C03599=1044.445,262.335,-106.667,171.686,39.912,157.590
C03600=1044.439,262.088,-106.637,171.684,39.910,157.589
C03601=1044.432,261.839,-106.607,171.681,39.908,157.589
C03602=1044.425,261.591,-106.577,171.677,39.906,157.588
C03603=1044.419,261.343,-106.548,171.675,39.903,157.587
C03604=1044.411,261.094,-106.518,171.672,39.901,157.587
C03605=1044.405,260.847,-106.488,171.669,39.898,157.586
C03606=1044.398,260.598,-106.459,171.666,39.896,157.586
C03607=1044.391,260.351,-106.429,171.663,39.894,157.585
C03608=1044.385,260.102,-106.400,171.661,39.892,157.584
C03609=1044.378,259.854,-106.370,171.658,39.889,157.584
C03610=1044.371,259.605,-106.341,171.654,39.887,157.583
C03611=1044.365,259.358,-106.311,171.652,39.885,157.583
C03612=1044.358,259.109,-106.282,171.649,39.882,157.582
C03613=1044.351,258.862,-106.252,171.646,39.880,157.581
C03614=1044.344,258.613,-106.222,171.643,39.878,157.581
C03615=1044.337,258.365,-106.194,171.640,39.876,157.580
C03616=1044.330,258.117,-106.164,171.638,39.873,157.580
C03617=1044.324,257.869,-106.135,171.635,39.871,157.579
C03618=1044.317,257.620,-106.105,171.632,39.868,157.578
C03619=1044.311,257.372,-106.076,171.629,39.866,157.578
C03620=1044.304,257.124,-106.047,171.626,39.864,157.577
C03621=1044.297,256.876,-106.016,171.624,39.862,157.577
C03622=1044.291,256.628,-105.987,171.621,39.859,157.576
C03623=1044.284,256.379,-105.958,171.618,39.857,157.575
C03624=1044.277,256.131,-105.928,171.615,39.855,157.575
C03625=1044.271,255.883,-105.899,171.612,39.852,157.574
C03626=1044.264,255.634,-105.870,171.610,39.850,157.573
C03627=1044.258,255.387,-105.840,171.607,39.848,157.573
C03628=1044.251,255.138,-105.811,171.604,39.845,157.572
C03629=1044.245,254.890,-105.782,171.602,39.843,157.572
C03630=1044.238,254.642,-105.753,171.598,39.841,157.571
C03631=1044.231,254.394,-105.723,171.595,39.838,157.570
C03632=1044.224,254.146,-105.694,171.593,39.836,157.570
C03633=1044.218,253.898,-105.665,171.590,39.834,157.569
C03634=1044.211,253.649,-105.636,171.588,39.831,157.569
C03635=1044.205,253.401,-105.606,171.585,39.829,157.568
C03636=1044.198,253.153,-105.577,171.583,39.827,157.567
C03637=1044.192,252.904,-105.547,171.579,39.824,157.567
C03638=1044.185,252.656,-105.518,171.576,39.822,157.566
C03639=1044.179,252.408,-105.489,171.574,39.820,157.566
C03640=1044.171,252.160,-105.460,171.571,39.817,157.565
C03641=1044.165,251.912,-105.431,171.568,39.815,157.564
C03642=1044.159,251.664,-105.402,171.566,39.812,157.564
C03643=1044.152,251.416,-105.373,171.563,39.810,157.563
C03644=1044.146,251.167,-105.343,171.561,39.808,157.563
C03645=1044.139,250.919,-105.314,171.557,39.806,157.562
C03646=1044.133,250.671,-105.285,171.554,39.803,157.561
C03647=1044.126,250.422,-105.256,171.552,39.801,157.561
C03648=1044.120,250.174,-105.227,171.549,39.798,157.560
C03649=1044.113,249.926,-105.198,171.546,39.796,157.560
C03650=1044.107,249.678,-105.169,171.544,39.794,157.559
C03651=1044.100,249.430,-105.140,171.541,39.791,157.558
C03652=1044.093,249.147,-105.106,171.539,39.789,157.558
C03653=1044.085,248.864,-105.074,171.535,39.786,157.557
C03654=1044.078,248.581,-105.040,171.532,39.784,157.556
C03655=1044.071,248.298,-105.008,171.530,39.781,157.556
C03656=1044.064,248.050,-104.978,171.527,39.778,157.555
C03657=1044.058,247.802,-104.949,171.523,39.776,157.554
C03658=1044.052,247.554,-104.920,171.521,39.773,157.554
C03659=1044.046,247.305,-104.891,171.518,39.771,157.553
C03660=1044.039,247.057,-104.862,171.515,39.769,157.553
C03661=1044.032,246.809,-104.834,171.513,39.767,157.552
C03662=1044.025,246.561,-104.804,171.510,39.764,157.551
C03663=1044.019,246.313,-104.775,171.508,39.762,157.551
C03664=1044.013,246.064,-104.746,171.505,39.759,157.550
C03665=1044.007,245.816,-104.718,171.502,39.757,157.550
C03666=1044.001,245.568,-104.689,171.500,39.755,157.549
C03667=1043.994,245.320,-104.661,171.497,39.752,157.548
C03668=1043.987,245.071,-104.631,171.495,39.750,157.548
C03669=1043.981,244.823,-104.602,171.492,39.747,157.547
C03670=1043.974,244.574,-104.574,171.489,39.745,157.547
C03671=1043.968,244.326,-104.545,171.487,39.743,157.546
C03672=1043.961,244.078,-104.516,171.484,39.741,157.545
C03673=1043.955,243.830,-104.489,171.482,39.738,157.545
C03674=1043.949,243.581,-104.460,171.479,39.736,157.544
C03675=1043.941,243.333,-104.431,171.477,39.734,157.544
C03676=1043.935,243.085,-104.402,171.474,39.731,157.543
C03677=1043.929,242.836,-104.373,171.471,39.729,157.542
C03678=1043.922,242.588,-104.345,171.469,39.726,157.542
C03679=1043.916,242.340,-104.317,171.466,39.724,157.541
C03680=1043.909,242.092,-104.288,171.464,39.722,157.541
C03681=1043.903,241.844,-104.259,171.461,39.720,157.540
C03682=1043.896,241.595,-104.231,171.458,39.717,157.539
C03683=1043.890,241.347,-104.202,171.456,39.715,157.539
C03684=1043.883,241.099,-104.173,171.453,39.713,157.538
C03685=1043.876,240.850,-104.145,171.451,39.711,157.538
C03686=1043.869,240.602,-104.117,171.448,39.708,157.537
C03687=1043.863,240.353,-104.088,171.445,39.706,157.537
C03688=1043.856,240.105,-104.060,171.443,39.704,157.536
C03689=1043.850,239.857,-104.032,171.440,39.701,157.535
C03690=1043.844,239.608,-104.004,171.438,39.699,157.535
C03691=1043.837,239.360,-103.976,171.435,39.696,157.534
C03692=1043.830,239.112,-103.948,171.432,39.694,157.534
C03693=1043.824,238.864,-103.919,171.430,39.692,157.533
C03694=1043.817,238.615,-103.891,171.427,39.690,157.532
C03695=1043.810,238.367,-103.863,171.425,39.687,157.532
C03696=1043.804,238.119,-103.834,171.422,39.685,157.531
C03697=1043.797,237.870,-103.806,171.420,39.683,157.531
C03698=1043.790,237.622,-103.778,171.417,39.680,157.530
C03699=1043.784,237.373,-103.749,171.415,39.678,157.530
C03700=1043.777,237.125,-103.721,171.413,39.676,157.529
C03701=1043.770,236.877,-103.693,171.410,39.674,157.528
C03702=1043.764,236.628,-103.665,171.408,39.671,157.528
C03703=1043.757,236.380,-103.636,171.405,39.669,157.527
C03704=1043.751,236.132,-103.609,171.403,39.667,157.527
C03705=1043.744,235.883,-103.581,171.400,39.665,157.526
C03706=1043.738,235.635,-103.553,171.397,39.662,157.526
C03707=1043.731,235.387,-103.524,171.395,39.660,157.525
C03708=1043.724,235.098,-103.492,171.392,39.657,157.524
C03709=1043.716,234.809,-103.459,171.390,39.655,157.524
C03710=1043.708,234.520,-103.427,171.386,39.652,157.523
C03711=1043.701,234.232,-103.394,171.383,39.649,157.522
C03712=1043.695,233.984,-103.366,171.381,39.647,157.522
C03713=1043.688,233.736,-103.339,171.378,39.645,157.521
C03714=1043.681,233.488,-103.310,171.377,39.642,157.521
C03715=1043.675,233.239,-103.282,171.374,39.640,157.520
C03716=1043.668,232.991,-103.254,171.371,39.638,157.519
C03717=1043.662,232.742,-103.226,171.369,39.635,157.519
C03718=1043.655,232.494,-103.199,171.366,39.633,157.518
C03719=1043.649,232.245,-103.170,171.364,39.631,157.518
C03720=1043.642,231.997,-103.142,171.361,39.629,157.517
C03721=1043.635,231.749,-103.114,171.359,39.626,157.517
C03722=1043.629,231.500,-103.086,171.357,39.624,157.516
C03723=1043.622,231.252,-103.059,171.354,39.622,157.515
C03724=1043.615,231.003,-103.031,171.352,39.619,157.515
C03725=1043.609,230.756,-103.004,171.349,39.617,157.514
C03726=1043.603,230.507,-102.976,171.347,39.615,157.514
C03727=1043.597,230.258,-102.947,171.344,39.613,157.513
C03728=1043.590,230.010,-102.920,171.342,39.610,157.513
C03729=1043.583,229.762,-102.892,171.340,39.608,157.512
C03730=1043.577,229.513,-102.864,171.337,39.606,157.512
C03731=1043.570,229.265,-102.837,171.335,39.603,157.511
C03732=1043.563,229.016,-102.809,171.332,39.601,157.510
C03733=1043.557,228.768,-102.781,171.330,39.599,157.510
C03734=1043.550,228.520,-102.754,171.327,39.597,157.509
C03735=1043.544,228.272,-102.726,171.325,39.594,157.509
C03736=1043.537,228.023,-102.698,171.323,39.592,157.508
C03737=1043.530,227.775,-102.671,171.321,39.590,157.508
C03738=1043.524,227.526,-102.644,171.318,39.587,157.507
C03739=1043.517,227.277,-102.616,171.315,39.585,157.506
C03740=1043.511,227.029,-102.588,171.313,39.583,157.506
C03741=1043.503,226.781,-102.561,171.310,39.581,157.505
C03742=1043.497,226.533,-102.534,171.309,39.578,157.505
C03743=1043.491,226.284,-102.506,171.306,39.576,157.504
C03744=1043.484,226.035,-102.479,171.304,39.574,157.504
C03745=1043.477,225.787,-102.451,171.301,39.571,157.503
C03746=1043.471,225.539,-102.423,171.298,39.569,157.502
C03747=1043.464,225.290,-102.396,171.297,39.567,157.502
C03748=1043.457,225.042,-102.368,171.294,39.564,157.501
C03749=1043.451,224.794,-102.342,171.292,39.562,157.501
C03750=1043.444,224.545,-102.314,171.289,39.560,157.500
C03751=1043.438,224.297,-102.286,171.287,39.558,157.500
C03752=1043.431,224.048,-102.259,171.285,39.555,157.499
C03753=1043.424,223.799,-102.232,171.283,39.553,157.498
C03754=1043.418,223.551,-102.204,171.280,39.551,157.498
C03755=1043.412,223.303,-102.177,171.277,39.548,157.497
C03756=1043.405,223.054,-102.150,171.275,39.546,157.497
C03757=1043.398,222.806,-102.122,171.273,39.544,157.496
C03758=1043.392,222.558,-102.095,171.271,39.541,157.496
C03759=1043.385,222.309,-102.068,171.268,39.539,157.495
C03760=1043.379,222.061,-102.040,171.266,39.537,157.495
C03761=1043.372,221.812,-102.013,171.264,39.534,157.494
C03762=1043.366,221.564,-101.986,171.262,39.532,157.493
C03763=1043.360,221.315,-101.958,171.259,39.530,157.493
C03764=1043.352,221.020,-101.926,171.256,39.527,157.492
C03765=1043.344,220.723,-101.893,171.254,39.524,157.491
C03766=1043.336,220.427,-101.861,171.251,39.522,157.491
C03767=1043.329,220.131,-101.829,171.248,39.519,157.490
C03768=1043.321,219.883,-101.802,171.246,39.517,157.490
C03769=1043.315,219.634,-101.775,171.243,39.514,157.489
C03770=1043.308,219.386,-101.748,171.242,39.512,157.488
C03771=1043.302,219.137,-101.721,171.239,39.510,157.488
C03772=1043.295,218.889,-101.693,171.237,39.507,157.487
C03773=1043.288,218.640,-101.667,171.234,39.505,157.487
C03774=1043.282,218.392,-101.639,171.233,39.503,157.486
C03775=1043.275,218.144,-101.613,171.230,39.500,157.486
C03776=1043.268,217.895,-101.586,171.227,39.498,157.485
C03777=1043.262,217.646,-101.558,171.226,39.496,157.485
C03778=1043.255,217.398,-101.532,171.223,39.493,157.484
C03779=1043.248,217.150,-101.504,171.221,39.492,157.484
C03780=1043.241,216.901,-101.478,171.218,39.489,157.483
C03781=1043.235,216.653,-101.451,171.217,39.487,157.482
C03782=1043.229,216.404,-101.424,171.214,39.485,157.482
C03783=1043.222,216.155,-101.397,171.212,39.483,157.481
C03784=1043.216,215.907,-101.370,171.210,39.480,157.481
C03785=1043.209,215.659,-101.343,171.208,39.478,157.480
C03786=1043.202,215.410,-101.316,171.205,39.476,157.480
C03787=1043.196,215.162,-101.290,171.203,39.473,157.479
C03788=1043.189,214.913,-101.263,171.201,39.471,157.479
C03789=1043.182,214.665,-101.236,171.198,39.469,157.478
C03790=1043.176,214.416,-101.209,171.197,39.466,157.477
C03791=1043.169,214.168,-101.182,171.194,39.464,157.477
C03792=1043.163,213.920,-101.156,171.192,39.462,157.476
C03793=1043.156,213.671,-101.129,171.190,39.459,157.476
C03794=1043.149,213.422,-101.102,171.188,39.457,157.475
C03795=1043.143,213.174,-101.075,171.185,39.455,157.475
C03796=1043.136,212.925,-101.048,171.184,39.452,157.474
C03797=1043.130,212.677,-101.022,171.181,39.450,157.473
C03798=1043.123,212.428,-100.995,171.178,39.448,157.473
C03799=1043.117,212.180,-100.968,171.177,39.445,157.472
C03800=1043.111,211.932,-100.941,171.174,39.442,157.472
C03801=1043.104,211.683,-100.915,171.172,39.440,157.471
C03802=1043.097,211.435,-100.889,171.170,39.438,157.471
C03803=1043.091,211.186,-100.862,171.168,39.435,157.470
C03804=1043.084,210.938,-100.835,171.166,39.433,157.469
C03805=1043.078,210.689,-100.808,171.163,39.431,157.469
C03806=1043.071,210.440,-100.781,171.161,39.429,157.468
C03807=1043.064,210.192,-100.755,171.160,39.427,157.468
C03808=1043.058,209.943,-100.728,171.157,39.424,157.467
C03809=1043.051,209.695,-100.702,171.154,39.422,157.467
C03810=1043.045,209.446,-100.675,171.153,39.420,157.466
C03811=1043.038,209.198,-100.649,171.150,39.417,157.466
C03812=1043.031,208.949,-100.623,171.149,39.415,157.465
C03813=1043.024,208.701,-100.596,171.146,39.413,157.465
C03814=1043.018,208.452,-100.570,171.144,39.410,157.464
C03815=1043.011,208.204,-100.543,171.142,39.408,157.463
C03816=1043.005,207.955,-100.517,171.140,39.406,157.463
C03817=1042.998,207.706,-100.490,171.138,39.403,157.462
C03818=1042.992,207.458,-100.464,171.136,39.401,157.462
C03819=1042.985,207.210,-100.438,171.133,39.399,157.461
C03820=1042.978,206.919,-100.407,171.130,39.396,157.461
C03821=1042.970,206.629,-100.376,171.129,39.393,157.460
C03822=1042.962,206.338,-100.346,171.126,39.391,157.459
C03823=1042.953,206.047,-100.315,171.123,39.388,157.459
C03824=1042.927,204.996,-100.208,170.852,39.286,157.429
C03825=1042.921,204.748,-100.183,170.849,39.284,157.428
C03826=1042.915,204.499,-100.157,170.846,39.282,157.428
C03827=1042.909,204.250,-100.133,170.843,39.281,157.428
C03828=1042.903,204.002,-100.108,170.840,39.279,157.427
C03829=1042.897,203.753,-100.082,170.837,39.278,157.427
C03830=1042.891,203.504,-100.057,170.835,39.276,157.426
C03831=1042.885,203.256,-100.032,170.831,39.275,157.426
C03832=1042.879,203.006,-100.007,170.829,39.273,157.426
C03833=1042.873,202.758,-99.982,170.826,39.271,157.425
C03834=1042.867,202.510,-99.957,170.823,39.270,157.425
C03835=1042.861,202.261,-99.932,170.820,39.269,157.424
C03836=1042.854,202.012,-99.908,170.817,39.267,157.424
C03837=1042.848,201.763,-99.882,170.814,39.265,157.423
C03838=1042.842,201.515,-99.857,170.812,39.264,157.423
C03839=1042.835,201.266,-99.832,170.808,39.263,157.423
C03840=1042.830,201.017,-99.807,170.806,39.261,157.422
C03841=1042.824,200.769,-99.782,170.803,39.259,157.422
C03842=1042.817,200.520,-99.758,170.800,39.258,157.422
C03843=1042.811,200.271,-99.733,170.797,39.256,157.421
C03844=1042.804,200.023,-99.708,170.794,39.255,157.421
C03845=1042.798,199.773,-99.683,170.791,39.254,157.420
C03846=1042.792,199.526,-99.659,170.789,39.252,157.420
C03847=1042.786,199.277,-99.634,170.787,39.251,157.420
C03848=1042.780,199.028,-99.609,170.783,39.249,157.419
C03849=1042.773,198.779,-99.585,170.781,39.248,157.419
C03850=1042.767,198.530,-99.559,170.777,39.247,157.419
C03851=1042.761,198.282,-99.536,170.775,39.245,157.418
C03852=1042.755,198.033,-99.510,170.772,39.244,157.418
C03853=1042.749,197.784,-99.486,170.769,39.242,157.417
C03854=1042.742,197.536,-99.461,170.766,39.241,157.417
C03855=1042.736,197.286,-99.436,170.764,39.239,157.417
C03856=1042.730,197.039,-99.412,170.760,39.238,157.416
C03857=1042.724,196.789,-99.387,170.758,39.237,157.416
C03858=1042.717,196.541,-99.363,170.755,39.235,157.415
C03859=1042.711,196.292,-99.338,170.752,39.234,157.415
C03860=1042.706,196.043,-99.314,170.749,39.232,157.415
C03861=1042.699,195.795,-99.289,170.747,39.231,157.414
C03862=1042.693,195.545,-99.265,170.744,39.229,157.414
C03863=1042.687,195.297,-99.241,170.741,39.228,157.414
C03864=1042.681,195.049,-99.216,170.739,39.227,157.413
C03865=1042.674,194.800,-99.191,170.735,39.225,157.413
C03866=1042.668,194.551,-99.166,170.733,39.224,157.413
C03867=1042.662,194.303,-99.142,170.730,39.222,157.412
C03868=1042.656,194.053,-99.118,170.727,39.221,157.412
C03869=1042.650,193.805,-99.093,170.725,39.220,157.411
C03870=1042.644,193.556,-99.069,170.722,39.219,157.411
C03871=1042.638,193.307,-99.044,170.719,39.217,157.411
C03872=1042.631,193.058,-99.020,170.716,39.216,157.410
C03873=1042.625,192.810,-98.995,170.714,39.214,157.410
C03874=1042.619,192.561,-98.971,170.711,39.213,157.410
C03875=1042.613,192.313,-98.947,170.708,39.211,157.409
C03876=1042.607,192.064,-98.923,170.706,39.210,157.409
C03877=1042.601,191.815,-98.898,170.702,39.209,157.409
C03878=1042.595,191.567,-98.874,170.700,39.207,157.408
C03879=1042.589,191.317,-98.849,170.697,39.206,157.408
C03880=1042.582,191.068,-98.825,170.694,39.205,157.407
C03881=1042.577,190.820,-98.801,170.692,39.203,157.407
C03882=1042.570,190.571,-98.776,170.689,39.202,157.407
C03883=1042.564,190.323,-98.752,170.686,39.200,157.406
C03884=1042.558,190.074,-98.728,170.684,39.199,157.406
C03885=1042.552,189.789,-98.700,170.680,39.198,157.406
C03886=1042.545,189.505,-98.672,170.677,39.196,157.405
C03887=1042.538,189.220,-98.645,170.675,39.194,157.405
C03888=1042.530,188.936,-98.617,170.671,39.193,157.404
C03889=1042.525,188.688,-98.593,170.669,39.191,157.404
C03890=1042.518,188.439,-98.569,170.666,39.190,157.404
C03891=1042.513,188.190,-98.544,170.663,39.189,157.403
C03892=1042.506,187.941,-98.520,170.661,39.188,157.403
C03893=1042.501,187.692,-98.496,170.658,39.186,157.403
C03894=1042.495,187.443,-98.472,170.655,39.185,157.402
C03895=1042.489,187.195,-98.448,170.653,39.183,157.402
C03896=1042.483,186.946,-98.424,170.650,39.182,157.402
C03897=1042.477,186.697,-98.400,170.647,39.181,157.401
C03898=1042.471,186.448,-98.375,170.645,39.179,157.401
C03899=1042.465,186.200,-98.351,170.642,39.178,157.401
C03900=1042.459,185.951,-98.327,170.639,39.177,157.400
C03901=1042.453,185.702,-98.303,170.637,39.175,157.400
C03902=1042.447,185.453,-98.279,170.634,39.174,157.399
C03903=1042.442,185.205,-98.255,170.631,39.173,157.399
C03904=1042.435,184.956,-98.231,170.629,39.172,157.399
C03905=1042.429,184.707,-98.207,170.626,39.170,157.398
C03906=1042.423,184.458,-98.182,170.624,39.169,157.398
C03907=1042.417,184.210,-98.159,170.621,39.167,157.398
C03908=1042.412,183.961,-98.134,170.619,39.166,157.397
C03909=1042.405,183.712,-98.110,170.616,39.165,157.397
C03910=1042.399,183.463,-98.087,170.613,39.163,157.397
C03911=1042.393,183.214,-98.063,170.611,39.162,157.396
C03912=1042.387,182.966,-98.040,170.608,39.161,157.396
C03913=1042.380,182.717,-98.016,170.605,39.160,157.396
C03914=1042.374,182.468,-97.993,170.603,39.159,157.395
C03915=1042.368,182.219,-97.969,170.600,39.158,157.395
C03916=1042.362,181.971,-97.945,170.598,39.157,157.395
C03917=1042.355,181.721,-97.922,170.595,39.156,157.395
C03918=1042.349,181.473,-97.898,170.592,39.154,157.394
C03919=1042.342,181.224,-97.874,170.590,39.153,157.394
C03920=1042.337,180.975,-97.851,170.587,39.152,157.394
C03921=1042.330,180.726,-97.827,170.584,39.151,157.393
C03922=1042.324,180.478,-97.803,170.582,39.150,157.393
C03923=1042.318,180.228,-97.780,170.580,39.149,157.393
C03924=1042.311,179.980,-97.757,170.576,39.148,157.392
C03925=1042.305,179.731,-97.734,170.574,39.146,157.392
C03926=1042.299,179.482,-97.710,170.572,39.145,157.392
C03927=1042.292,179.233,-97.686,170.569,39.144,157.392
C03928=1042.286,178.985,-97.663,170.566,39.143,157.391
C03929=1042.280,178.736,-97.639,170.564,39.141,157.391
C03930=1042.274,178.487,-97.616,170.561,39.140,157.391
C03931=1042.268,178.238,-97.593,170.558,39.139,157.390
C03932=1042.262,177.989,-97.569,170.556,39.138,157.390
C03933=1042.255,177.741,-97.546,170.554,39.137,157.390
C03934=1042.248,177.491,-97.523,170.551,39.136,157.389
C03935=1042.242,177.243,-97.499,170.548,39.135,157.389
C03936=1042.237,176.994,-97.476,170.546,39.134,157.389
C03937=1042.230,176.745,-97.452,170.543,39.133,157.388
C03938=1042.224,176.496,-97.429,170.540,39.132,157.388
C03939=1042.218,176.248,-97.406,170.538,39.131,157.388
C03940=1042.212,175.998,-97.382,170.536,39.129,157.388
C03941=1042.206,175.750,-97.359,170.533,39.128,157.387
C03942=1042.200,175.500,-97.335,170.530,39.127,157.387
C03943=1042.193,175.253,-97.312,170.528,39.126,157.387
C03944=1042.187,175.004,-97.289,170.526,39.125,157.386
C03945=1042.181,174.754,-97.266,170.522,39.123,157.386
C03946=1042.175,174.506,-97.242,170.520,39.122,157.386
C03947=1042.169,174.257,-97.219,170.518,39.121,157.385
C03948=1042.163,174.009,-97.196,170.516,39.120,157.385
C03949=1042.155,173.723,-97.170,170.512,39.119,157.385
C03950=1042.149,173.438,-97.143,170.510,39.118,157.385
C03951=1042.142,173.153,-97.116,170.507,39.116,157.384
C03952=1042.135,172.869,-97.090,170.503,39.115,157.384
C03953=1042.129,172.620,-97.066,170.501,39.114,157.383
C03954=1042.122,172.371,-97.043,170.499,39.113,157.383
C03955=1042.117,172.122,-97.020,170.497,39.112,157.383
C03956=1042.110,171.874,-96.997,170.494,39.111,157.383
C03957=1042.104,171.625,-96.974,170.491,39.110,157.382
C03958=1042.098,171.375,-96.951,170.489,39.109,157.382
C03959=1042.092,171.126,-96.928,170.487,39.108,157.382
C03960=1042.086,170.878,-96.904,170.484,39.107,157.381
C03961=1042.080,170.629,-96.881,170.481,39.105,157.381
C03962=1042.074,170.380,-96.858,170.479,39.104,157.381
C03963=1042.067,170.131,-96.836,170.477,39.103,157.381
C03964=1042.061,169.883,-96.812,170.474,39.102,157.380
C03965=1042.056,169.634,-96.789,170.472,39.100,157.380
C03966=1042.049,169.384,-96.766,170.470,39.099,157.380
C03967=1042.044,169.135,-96.743,170.466,39.098,157.379
C03968=1042.038,168.887,-96.720,170.464,39.097,157.379
C03969=1042.031,168.639,-96.697,170.462,39.096,157.379
C03970=1042.025,168.390,-96.674,170.460,39.095,157.378
C03971=1042.020,168.141,-96.651,170.457,39.094,157.378
C03972=1042.013,167.891,-96.627,170.454,39.093,157.378
C03973=1042.008,167.642,-96.604,170.452,39.092,157.378
C03974=1042.002,167.393,-96.582,170.449,39.091,157.377
C03975=1041.995,167.145,-96.559,170.447,39.089,157.377
C03976=1041.989,166.897,-96.536,170.445,39.088,157.377
C03977=1041.984,166.648,-96.513,170.443,39.087,157.376
C03978=1041.978,166.399,-96.490,170.439,39.086,157.376
C03979=1041.972,166.149,-96.466,170.437,39.085,157.376
C03980=1041.965,165.901,-96.444,170.435,39.084,157.376
C03981=1041.959,165.652,-96.421,170.433,39.083,157.375
C03982=1041.954,165.403,-96.398,170.430,39.082,157.375
C03983=1041.948,165.154,-96.375,170.428,39.081,157.375
C03984=1041.942,164.905,-96.352,170.426,39.079,157.374
C03985=1041.936,164.656,-96.330,170.423,39.078,157.374
C03986=1041.930,164.408,-96.307,170.420,39.077,157.374
C03987=1041.924,164.159,-96.284,170.418,39.076,157.373
C03988=1041.919,163.910,-96.261,170.416,39.075,157.373
C03989=1041.913,163.661,-96.238,170.414,39.074,157.373
C03990=1041.906,163.412,-96.215,170.411,39.073,157.373
C03991=1041.900,163.163,-96.192,170.409,39.072,157.372
C03992=1041.894,162.914,-96.169,170.407,39.071,157.372
C03993=1041.889,162.665,-96.147,170.403,39.070,157.372
C03994=1041.883,162.416,-96.124,170.401,39.068,157.371
C03995=1041.876,162.167,-96.101,170.399,39.067,157.371
C03996=1041.871,161.918,-96.078,170.397,39.066,157.371
C03997=1041.865,161.670,-96.055,170.394,39.065,157.371
C03998=1041.859,161.421,-96.032,170.392,39.064,157.370
C03999=1041.853,161.172,-96.010,170.390,39.063,157.370
C04000=1041.847,160.923,-95.988,170.388,39.062,157.370
C04001=1041.842,160.674,-95.965,170.385,39.061,157.369
C04002=1041.836,160.425,-95.942,170.383,39.060,157.369
C04003=1041.829,160.176,-95.920,170.380,39.059,157.369
C04004=1041.824,159.927,-95.897,170.378,39.058,157.369
C04005=1041.817,159.678,-95.875,170.375,39.057,157.368
C04006=1041.812,159.429,-95.852,170.373,39.056,157.368
C04007=1041.805,159.181,-95.830,170.371,39.055,157.368
C04008=1041.799,158.932,-95.807,170.369,39.054,157.368
C04009=1041.793,158.683,-95.785,170.367,39.053,157.367
C04010=1041.787,158.434,-95.763,170.364,39.052,157.367
C04011=1041.781,158.185,-95.740,170.361,39.051,157.367
C04012=1041.775,157.936,-95.718,170.359,39.050,157.367
C04013=1041.766,157.610,-95.689,170.357,39.049,157.366
C04014=1041.758,157.283,-95.659,170.353,39.048,157.366
C04015=1041.751,156.956,-95.630,170.350,39.046,157.366
C04016=1041.742,156.630,-95.601,170.347,39.045,157.365
C04017=1041.737,156.381,-95.578,170.344,39.044,157.365
C04018=1041.730,156.132,-95.556,170.342,39.043,157.365
C04019=1041.724,155.884,-95.534,170.340,39.042,157.364
C04020=1041.718,155.634,-95.511,170.338,39.041,157.364
C04021=1041.712,155.385,-95.489,170.335,39.040,157.364
C04022=1041.706,155.136,-95.467,170.333,39.039,157.364
C04023=1041.700,154.887,-95.444,170.331,39.038,157.363
C04024=1041.694,154.639,-95.422,170.328,39.037,157.363
C04025=1041.687,154.390,-95.400,170.325,39.036,157.363
C04026=1041.682,154.141,-95.377,170.323,39.035,157.363
C04027=1041.676,153.891,-95.356,170.321,39.035,157.362
C04028=1041.669,153.643,-95.334,170.319,39.033,157.362
C04029=1041.663,153.394,-95.312,170.317,39.032,157.362
C04030=1041.657,153.145,-95.289,170.314,39.032,157.362
C04031=1041.651,152.896,-95.267,170.312,39.031,157.361
C04032=1041.645,152.647,-95.245,170.310,39.030,157.361
C04033=1041.638,152.398,-95.223,170.308,39.028,157.361
C04034=1041.632,152.149,-95.201,170.306,39.028,157.361
C04035=1041.627,151.900,-95.179,170.303,39.027,157.360
C04036=1041.621,151.651,-95.157,170.300,39.026,157.360
C04037=1041.614,151.403,-95.135,170.298,39.025,157.360
C04038=1041.608,151.153,-95.113,170.296,39.024,157.360
C04039=1041.602,150.905,-95.091,170.293,39.023,157.359
C04040=1041.596,150.655,-95.069,170.291,39.023,157.359
C04041=1041.590,150.407,-95.047,170.289,39.021,157.359
C04042=1041.584,150.157,-95.025,170.287,39.020,157.359
C04043=1041.578,149.908,-95.003,170.284,39.019,157.358
C04044=1041.571,149.660,-94.981,170.282,39.019,157.358
C04045=1041.566,149.410,-94.959,170.280,39.018,157.358
C04046=1041.560,149.162,-94.937,170.278,39.016,157.358
C04047=1041.554,148.913,-94.915,170.276,39.016,157.357
C04048=1041.548,148.664,-94.893,170.273,39.015,157.357
C04049=1041.542,148.436,-94.873,170.271,39.014,157.357
C04050=1041.536,148.207,-94.853,170.269,39.013,157.357
C04051=1041.531,147.978,-94.833,170.267,39.013,157.357
C04052=1041.525,147.750,-94.813,170.265,39.012,157.356
C04053=1041.519,147.521,-94.792,170.262,39.010,157.356
C04054=1041.514,147.293,-94.773,170.260,39.010,157.356
C04055=1041.508,147.065,-94.753,170.259,39.009,157.356
C04056=1041.503,146.837,-94.733,170.257,39.008,157.355
C04057=1041.497,146.588,-94.712,170.255,39.007,157.355
C04058=1041.490,146.338,-94.690,170.252,39.007,157.355
C04059=1041.484,146.089,-94.668,170.250,39.006,157.355
C04060=1041.478,145.841,-94.646,170.247,39.005,157.355
C04061=1041.472,145.591,-94.624,170.245,39.004,157.354
C04062=1041.466,145.343,-94.603,170.243,39.004,157.354
C04063=1041.460,145.094,-94.581,170.240,39.002,157.354
C04064=1041.454,144.845,-94.560,170.238,39.001,157.354
C04065=1041.448,144.595,-94.538,170.236,39.001,157.353
C04066=1041.441,144.347,-94.516,170.234,39.000,157.353
C04067=1041.435,144.098,-94.494,170.232,38.999,157.353
C04068=1041.429,143.849,-94.473,170.229,38.998,157.353
C04069=1041.423,143.600,-94.451,170.227,38.997,157.352
C04070=1041.417,143.351,-94.430,170.225,38.996,157.352
C04071=1041.410,143.102,-94.409,170.223,38.995,157.352
C04072=1041.404,142.853,-94.387,170.221,38.995,157.352
C04073=1041.398,142.604,-94.366,170.218,38.994,157.351
C04074=1041.392,142.355,-94.344,170.216,38.993,157.351
C04075=1041.386,142.106,-94.322,170.214,38.992,157.351
C04076=1041.380,141.856,-94.301,170.212,38.991,157.351
C04077=1041.373,141.571,-94.276,170.209,38.990,157.351
C04078=1041.366,141.286,-94.250,170.206,38.989,157.350
C04079=1041.359,141.000,-94.227,170.204,38.988,157.350
C04080=1041.352,140.714,-94.201,170.202,38.987,157.350
C04081=1041.346,140.465,-94.180,170.200,38.987,157.350
C04082=1041.340,140.217,-94.159,170.197,38.986,157.349
C04083=1041.334,139.967,-94.137,170.195,38.984,157.349
C04084=1041.328,139.718,-94.115,170.193,38.984,157.349
C04085=1041.322,139.469,-94.094,170.191,38.983,157.349
C04086=1041.315,139.221,-94.073,170.189,38.982,157.348
C04087=1041.309,138.972,-94.051,170.186,38.981,157.348
C04088=1041.303,138.722,-94.030,170.184,38.981,157.348
C04089=1041.297,138.473,-94.009,170.182,38.980,157.348
C04090=1041.291,138.224,-93.988,170.180,38.979,157.348
C04091=1041.285,137.975,-93.966,170.177,38.978,157.347
C04092=1041.279,137.726,-93.945,170.175,38.977,157.347
C04093=1041.272,137.477,-93.923,170.173,38.976,157.347
C04094=1041.266,137.229,-93.903,170.171,38.976,157.347
C04095=1041.260,136.979,-93.881,170.169,38.975,157.346
C04096=1041.254,136.730,-93.860,170.167,38.974,157.346
C04097=1041.249,136.481,-93.839,170.164,38.973,157.346
C04098=1041.242,136.232,-93.818,170.162,38.973,157.346
C04099=1041.236,135.983,-93.796,170.160,38.971,157.345
C04100=1041.229,135.734,-93.774,170.158,38.971,157.345
C04101=1041.223,135.485,-93.754,170.156,38.970,157.345
C04102=1041.217,135.236,-93.733,170.153,38.969,157.345
C04103=1041.211,134.987,-93.711,170.151,38.968,157.345
C04104=1041.205,134.738,-93.691,170.149,38.968,157.344
C04105=1041.199,134.489,-93.669,170.147,38.966,157.344
C04106=1041.193,134.239,-93.648,170.145,38.966,157.344
C04107=1041.186,133.991,-93.627,170.142,38.965,157.344
C04108=1041.180,133.742,-93.606,170.140,38.964,157.344
C04109=1041.174,133.492,-93.585,170.138,38.963,157.343
C04110=1041.168,133.244,-93.564,170.136,38.963,157.343
C04111=1041.162,132.995,-93.542,170.134,38.962,157.343
C04112=1041.156,132.745,-93.521,170.131,38.961,157.343
C04113=1041.150,132.497,-93.501,170.129,38.961,157.343
C04114=1041.144,132.247,-93.479,170.127,38.959,157.342
C04115=1041.138,131.999,-93.458,170.125,38.959,157.342
C04116=1041.131,131.749,-93.438,170.123,38.958,157.342
C04117=1041.125,131.500,-93.416,170.121,38.957,157.342
C04118=1041.120,131.252,-93.395,170.118,38.956,157.341
C04119=1041.113,131.002,-93.374,170.116,38.956,157.341
C04120=1041.107,130.753,-93.353,170.114,38.955,157.341
C04121=1041.101,130.504,-93.333,170.112,38.954,157.341
C04122=1041.094,130.255,-93.312,170.110,38.954,157.341
C04123=1041.088,130.005,-93.291,170.107,38.952,157.340
C04124=1041.082,129.757,-93.270,170.105,38.952,157.340
C04125=1041.075,129.508,-93.250,170.103,38.951,157.340
C04126=1041.069,129.259,-93.228,170.101,38.950,157.340
C04127=1041.063,129.010,-93.208,170.099,38.950,157.340
C04128=1041.056,128.761,-93.187,170.097,38.949,157.339
C04129=1041.050,128.511,-93.166,170.095,38.948,157.339
C04130=1041.044,128.263,-93.146,170.093,38.948,157.339
C04131=1041.038,128.013,-93.125,170.091,38.947,157.339
C04132=1041.032,127.765,-93.104,170.089,38.946,157.339
C04133=1041.025,127.515,-93.084,170.087,38.945,157.338
C04134=1041.018,127.266,-93.063,170.085,38.945,157.338
C04135=1041.013,127.017,-93.042,170.082,38.944,157.338
C04136=1041.006,126.768,-93.021,170.080,38.943,157.338
C04137=1041.000,126.520,-93.001,170.078,38.943,157.338
C04138=1040.994,126.270,-92.979,170.076,38.942,157.337
C04139=1040.988,126.021,-92.959,170.074,38.941,157.337
C04140=1040.982,125.772,-92.939,170.071,38.941,157.337
C04141=1040.975,125.486,-92.915,170.069,38.940,157.337
C04142=1040.968,125.200,-92.891,170.066,38.939,157.337
C04143=1040.961,124.915,-92.867,170.064,38.938,157.336
C04144=1040.953,124.628,-92.844,170.062,38.938,157.336
C04145=1040.947,124.380,-92.823,170.059,38.936,157.336
C04146=1040.940,124.130,-92.803,170.057,38.936,157.336
C04147=1040.935,123.881,-92.782,170.055,38.935,157.335
C04148=1040.928,123.632,-92.761,170.053,38.934,157.335
C04149=1040.922,123.384,-92.741,170.051,38.934,157.335
C04150=1040.916,123.134,-92.720,170.049,38.933,157.335
C04151=1040.910,122.886,-92.700,170.046,38.932,157.335
C04152=1040.904,122.636,-92.679,170.044,38.932,157.335
C04153=1040.898,122.387,-92.659,170.043,38.930,157.334
C04154=1040.891,122.138,-92.638,170.041,38.930,157.334
C04155=1040.885,121.889,-92.618,170.039,38.929,157.334
C04156=1040.880,121.639,-92.597,170.036,38.928,157.334
C04157=1040.874,121.391,-92.577,170.034,38.928,157.334
C04158=1040.867,121.142,-92.556,170.032,38.927,157.333
C04159=1040.861,120.893,-92.536,170.030,38.926,157.333
C04160=1040.855,120.643,-92.515,170.028,38.926,157.333
C04161=1040.849,120.394,-92.495,170.026,38.924,157.333
C04162=1040.842,120.145,-92.474,170.023,38.924,157.332
C04163=1040.837,119.896,-92.454,170.021,38.923,157.332
C04164=1040.830,119.647,-92.433,170.019,38.922,157.332
C04165=1040.824,119.398,-92.413,170.018,38.922,157.332
C04166=1040.819,119.149,-92.392,170.016,38.921,157.332
C04167=1040.812,118.900,-92.372,170.014,38.920,157.331
C04168=1040.806,118.651,-92.352,170.011,38.920,157.331
C04169=1040.799,118.402,-92.331,170.009,38.918,157.331
C04170=1040.794,118.152,-92.311,170.007,38.918,157.331
C04171=1040.787,117.903,-92.290,170.005,38.917,157.331
C04172=1040.781,117.655,-92.270,170.003,38.916,157.330
C04173=1040.776,117.406,-92.249,170.000,38.916,157.330
C04174=1040.769,117.156,-92.229,169.998,38.915,157.330
C04175=1040.763,116.907,-92.209,169.997,38.914,157.330
C04176=1040.757,116.658,-92.189,169.995,38.914,157.330
C04177=1040.751,116.409,-92.168,169.993,38.912,157.329
C04178=1040.745,116.160,-92.148,169.991,38.912,157.329
C04179=1040.739,115.910,-92.128,169.988,38.911,157.329
C04180=1040.733,115.661,-92.108,169.986,38.910,157.329
C04181=1040.727,115.413,-92.087,169.984,38.910,157.329
C04182=1040.721,115.163,-92.066,169.982,38.909,157.328
C04183=1040.715,114.915,-92.046,169.980,38.908,157.328
C04184=1040.709,114.665,-92.025,169.979,38.908,157.328
C04185=1040.703,114.416,-92.005,169.976,38.906,157.328
C04186=1040.697,114.167,-91.985,169.974,38.906,157.328
C04187=1040.690,113.918,-91.965,169.972,38.905,157.327
C04188=1040.685,113.669,-91.945,169.970,38.904,157.327
C04189=1040.679,113.420,-91.925,169.968,38.904,157.327
C04190=1040.672,113.170,-91.904,169.965,38.903,157.327
C04191=1040.666,112.921,-91.884,169.963,38.902,157.327
C04192=1040.660,112.673,-91.864,169.962,38.902,157.326
C04193=1040.654,112.423,-91.844,169.960,38.900,157.326
C04194=1040.648,112.174,-91.824,169.958,38.900,157.326
C04195=1040.642,111.925,-91.804,169.956,38.899,157.326
C04196=1040.636,111.675,-91.785,169.953,38.899,157.326
C04197=1040.630,111.426,-91.765,169.951,38.898,157.325
C04198=1040.624,111.178,-91.745,169.949,38.897,157.325
C04199=1040.617,110.928,-91.724,169.947,38.897,157.325
C04200=1040.611,110.679,-91.704,169.945,38.896,157.325
C04201=1040.604,110.430,-91.684,169.943,38.895,157.325
C04202=1040.598,110.181,-91.664,169.941,38.895,157.325
C04203=1040.592,109.932,-91.645,169.939,38.894,157.324
C04204=1040.585,109.682,-91.625,169.937,38.894,157.324
C04205=1040.579,109.396,-91.602,169.935,38.892,157.324
C04206=1040.571,109.111,-91.580,169.932,38.892,157.324
C04207=1040.565,108.825,-91.557,169.930,38.892,157.324
C04208=1040.557,108.539,-91.535,169.927,38.890,157.323
C04209=1040.551,108.289,-91.514,169.925,38.890,157.323
C04210=1040.545,108.041,-91.494,169.923,38.889,157.323
C04211=1040.539,107.792,-91.474,169.921,38.889,157.323
C04212=1040.532,107.542,-91.454,169.919,38.888,157.323
C04213=1040.526,107.293,-91.435,169.918,38.887,157.322
C04214=1040.520,107.044,-91.415,169.916,38.887,157.322
C04215=1040.513,106.795,-91.395,169.913,38.886,157.322
C04216=1040.507,106.545,-91.376,169.911,38.886,157.322
C04217=1040.501,106.297,-91.356,169.909,38.884,157.322
C04218=1040.495,106.048,-91.336,169.907,38.884,157.322
C04219=1040.489,105.798,-91.316,169.905,38.883,157.321
C04220=1040.482,105.549,-91.297,169.903,38.883,157.321
C04221=1040.476,105.300,-91.277,169.901,38.882,157.321
C04222=1040.470,105.051,-91.257,169.899,38.881,157.321
C04223=1040.464,104.801,-91.237,169.897,38.881,157.321
C04224=1040.458,104.553,-91.217,169.895,38.880,157.321
C04225=1040.451,104.304,-91.198,169.893,38.880,157.320
C04226=1040.445,104.054,-91.178,169.891,38.879,157.320
C04227=1040.439,103.805,-91.158,169.888,38.878,157.320
C04228=1040.433,103.556,-91.139,169.886,38.878,157.320
C04229=1040.427,103.307,-91.119,169.885,38.877,157.320
C04230=1040.421,103.058,-91.099,169.883,38.876,157.319
C04231=1040.414,102.808,-91.080,169.881,38.875,157.319
C04232=1040.408,102.559,-91.060,169.879,38.875,157.319
C04233=1040.403,102.310,-91.041,169.877,38.874,157.319
C04234=1040.397,102.061,-91.021,169.874,38.873,157.319
C04235=1040.391,101.812,-91.001,169.872,38.873,157.318
C04236=1040.384,101.563,-90.982,169.871,38.872,157.318
C04237=1040.378,101.314,-90.962,169.869,38.872,157.318
C04238=1040.372,101.064,-90.943,169.867,38.870,157.318
C04239=1040.366,100.815,-90.923,169.865,38.870,157.318
C04240=1040.360,100.566,-90.904,169.862,38.869,157.318
C04241=1040.353,100.317,-90.884,169.860,38.869,157.317
C04242=1040.347,100.067,-90.865,169.858,38.868,157.317
C04243=1040.340,99.819,-90.845,169.856,38.867,157.317
C04244=1040.335,99.569,-90.826,169.855,38.867,157.317
C04245=1040.329,99.321,-90.806,169.853,38.866,157.317
C04246=1040.322,99.071,-90.787,169.850,38.866,157.317
C04247=1040.316,98.822,-90.767,169.848,38.865,157.316
C04248=1040.309,98.573,-90.749,169.846,38.865,157.316
C04249=1040.304,98.323,-90.729,169.844,38.864,157.316
C04250=1040.297,98.075,-90.710,169.842,38.863,157.316
C04251=1040.291,97.825,-90.690,169.840,38.862,157.316
C04252=1040.284,97.576,-90.671,169.839,38.862,157.316
C04253=1040.278,97.327,-90.652,169.836,38.861,157.315
C04254=1040.272,97.078,-90.633,169.834,38.861,157.315
C04255=1040.266,96.829,-90.613,169.832,38.860,157.315
C04256=1040.259,96.579,-90.594,169.830,38.860,157.315
C04257=1040.253,96.330,-90.575,169.828,38.859,157.315
C04258=1040.246,96.081,-90.556,169.826,38.858,157.314
C04259=1040.241,95.832,-90.536,169.824,38.858,157.314
C04260=1040.235,95.582,-90.517,169.822,38.857,157.314
C04261=1040.228,95.334,-90.498,169.820,38.857,157.314
C04262=1040.223,95.084,-90.478,169.818,38.856,157.314
C04263=1040.216,94.835,-90.460,169.816,38.856,157.314
C04264=1040.210,94.586,-90.439,169.814,38.854,157.313
C04265=1040.203,94.337,-90.421,169.812,38.854,157.313
C04266=1040.197,94.087,-90.402,169.809,38.853,157.313
C04267=1040.191,93.839,-90.382,169.808,38.853,157.313
C04268=1040.185,93.589,-90.363,169.806,38.852,157.313
C04269=1040.178,93.303,-90.341,169.804,38.851,157.313
C04270=1040.170,93.017,-90.319,169.802,38.851,157.312
C04271=1040.163,92.731,-90.297,169.799,38.850,157.312
C04272=1040.156,92.445,-90.275,169.796,38.849,157.312
C04273=1040.150,92.196,-90.256,169.794,38.849,157.312
C04274=1040.144,91.947,-90.237,169.793,38.848,157.312
C04275=1040.138,91.697,-90.218,169.791,38.847,157.312
C04276=1040.132,91.448,-90.199,169.789,38.847,157.311
C04277=1040.126,91.199,-90.179,169.787,38.846,157.311
C04278=1040.119,90.950,-90.161,169.785,38.845,157.311
C04279=1040.113,90.701,-90.141,169.782,38.845,157.311
C04280=1040.107,90.452,-90.123,169.781,38.844,157.311
C04281=1040.101,90.202,-90.103,169.779,38.844,157.310
C04282=1040.095,89.953,-90.085,169.777,38.843,157.310
C04283=1040.088,89.705,-90.065,169.775,38.843,157.310
C04284=1040.083,89.455,-90.046,169.773,38.842,157.310
C04285=1040.076,89.205,-90.027,169.771,38.842,157.310
C04286=1040.069,88.956,-90.009,169.769,38.841,157.310
C04287=1040.063,88.707,-89.990,169.766,38.840,157.309
C04288=1040.057,88.458,-89.971,169.765,38.839,157.309
C04289=1040.051,88.209,-89.952,169.763,38.839,157.309
C04290=1040.044,87.959,-89.933,169.761,38.838,157.309
C04291=1040.038,87.710,-89.915,169.759,38.838,157.309
C04292=1040.031,87.461,-89.896,169.757,38.837,157.309
C04293=1040.026,87.212,-89.877,169.754,38.837,157.309
C04294=1040.019,86.963,-89.858,169.752,38.836,157.308
C04295=1040.013,86.713,-89.840,169.750,38.836,157.308
C04296=1040.006,86.464,-89.821,169.749,38.835,157.308
C04297=1040.001,86.215,-89.802,169.747,38.835,157.308
C04298=1039.994,85.966,-89.783,169.745,38.834,157.308
C04299=1039.988,85.717,-89.764,169.743,38.834,157.308
C04300=1039.981,85.468,-89.746,169.741,38.833,157.307
C04301=1039.975,85.218,-89.727,169.738,38.833,157.307
C04302=1039.969,84.969,-89.708,169.736,38.832,157.307
C04303=1039.963,84.720,-89.689,169.735,38.832,157.307
C04304=1039.956,84.471,-89.671,169.733,38.830,157.307
C04305=1039.950,84.222,-89.652,169.731,38.830,157.307
C04306=1039.944,83.973,-89.633,169.729,38.829,157.306
C04307=1039.938,83.723,-89.614,169.727,38.829,157.306
C04308=1039.931,83.474,-89.595,169.724,38.828,157.306
C04309=1039.925,83.224,-89.577,169.722,38.828,157.306
C04310=1039.919,82.975,-89.559,169.721,38.827,157.306
C04311=1039.912,82.726,-89.540,169.719,38.827,157.306
C04312=1039.907,82.477,-89.521,169.717,38.826,157.306
C04313=1039.900,82.227,-89.502,169.715,38.826,157.305
C04314=1039.894,81.978,-89.484,169.713,38.825,157.305
C04315=1039.887,81.729,-89.465,169.710,38.824,157.305
C04316=1039.881,81.480,-89.446,169.709,38.824,157.305
C04317=1039.876,81.230,-89.428,169.707,38.823,157.305
C04318=1039.869,80.981,-89.409,169.705,38.822,157.304
C04319=1039.863,80.732,-89.390,169.703,38.822,157.304
C04320=1039.857,80.483,-89.372,169.701,38.821,157.304
C04321=1039.851,80.234,-89.353,169.699,38.821,157.304
C04322=1039.844,79.985,-89.335,169.696,38.820,157.304
C04323=1039.839,79.735,-89.316,169.695,38.820,157.304
C04324=1039.832,79.486,-89.298,169.693,38.819,157.303
C04325=1039.826,79.237,-89.279,169.691,38.818,157.303
C04326=1039.819,78.988,-89.260,169.689,38.818,157.303
C04327=1039.813,78.739,-89.242,169.687,38.817,157.303
C04328=1039.807,78.489,-89.224,169.685,38.817,157.303
C04329=1039.801,78.239,-89.205,169.683,38.816,157.303
C04330=1039.795,77.991,-89.186,169.681,38.816,157.303
C04331=1039.789,77.741,-89.168,169.679,38.815,157.302
C04332=1039.783,77.492,-89.150,169.677,38.815,157.302
C04333=1039.775,77.206,-89.129,169.675,38.814,157.302
C04334=1039.768,76.920,-89.107,169.673,38.813,157.302
C04335=1039.761,76.634,-89.086,169.671,38.812,157.302
C04336=1039.754,76.347,-89.065,169.668,38.812,157.302
C04337=1039.747,76.098,-89.047,169.666,38.811,157.301
C04338=1039.741,75.849,-89.028,169.664,38.811,157.301
C04339=1039.735,75.600,-89.010,169.662,38.810,157.301
C04340=1039.729,75.351,-88.992,169.660,38.810,157.301
C04341=1039.722,75.102,-88.975,169.658,38.809,157.301
C04342=1039.716,74.853,-88.956,169.656,38.809,157.301
C04343=1039.709,74.603,-88.937,169.654,38.808,157.300
C04344=1039.703,74.354,-88.919,169.652,38.808,157.300
C04345=1039.697,74.105,-88.901,169.650,38.807,157.300
C04346=1039.691,73.855,-88.883,169.648,38.807,157.300
C04347=1039.685,73.606,-88.864,169.646,38.806,157.300
C04348=1039.678,73.357,-88.846,169.644,38.806,157.300
C04349=1039.672,73.108,-88.828,169.642,38.805,157.300
C04350=1039.666,72.858,-88.809,169.640,38.805,157.299
C04351=1039.660,72.609,-88.791,169.638,38.804,157.299
C04352=1039.652,72.360,-88.773,169.636,38.803,157.299
C04353=1039.647,72.111,-88.756,169.634,38.803,157.299
C04354=1039.641,71.862,-88.737,169.632,38.802,157.299
C04355=1039.634,71.612,-88.719,169.630,38.802,157.299
C04356=1039.628,71.363,-88.700,169.628,38.801,157.298
C04357=1039.622,71.113,-88.683,169.626,38.801,157.298
C04358=1039.615,70.864,-88.664,169.625,38.800,157.298
C04359=1039.610,70.615,-88.646,169.622,38.800,157.298
C04360=1039.603,70.366,-88.628,169.620,38.799,157.298
C04361=1039.597,70.116,-88.610,169.618,38.799,157.298
C04362=1039.590,69.867,-88.592,169.616,38.798,157.298
C04363=1039.585,69.618,-88.574,169.614,38.798,157.297
C04364=1039.579,69.368,-88.556,169.613,38.797,157.297
C04365=1039.572,69.119,-88.538,169.611,38.797,157.297
C04366=1039.565,68.870,-88.520,169.609,38.796,157.297
C04367=1039.559,68.621,-88.502,169.606,38.796,157.297
C04368=1039.553,68.372,-88.484,169.604,38.795,157.297
C04369=1039.547,68.122,-88.466,169.602,38.794,157.297
C04370=1039.540,67.873,-88.448,169.600,38.794,157.296
C04371=1039.534,67.623,-88.430,169.598,38.793,157.296
C04372=1039.528,67.374,-88.412,169.597,38.793,157.296
C04373=1039.521,67.126,-88.394,169.595,38.792,157.296
C04374=1039.515,66.876,-88.377,169.593,38.792,157.296
C04375=1039.509,66.626,-88.359,169.590,38.791,157.296
C04376=1039.503,66.377,-88.340,169.588,38.791,157.295
C04377=1039.496,66.128,-88.323,169.586,38.790,157.295
C04378=1039.490,65.879,-88.305,169.584,38.790,157.295
C04379=1039.484,65.629,-88.286,169.583,38.789,157.295
C04380=1039.477,65.380,-88.269,169.581,38.789,157.295
C04381=1039.471,65.131,-88.251,169.579,38.788,157.295
C04382=1039.465,64.882,-88.233,169.576,38.788,157.295
C04383=1039.458,64.632,-88.215,169.574,38.787,157.294
C04384=1039.453,64.383,-88.198,169.572,38.787,157.294
C04385=1039.447,64.134,-88.180,169.570,38.786,157.294
C04386=1039.440,63.884,-88.163,169.568,38.786,157.294
C04387=1039.433,63.635,-88.144,169.567,38.785,157.294
C04388=1039.426,63.386,-88.127,169.565,38.785,157.294
C04389=1039.421,63.137,-88.109,169.563,38.785,157.294
C04390=1039.414,62.887,-88.092,169.561,38.784,157.293
C04391=1039.407,62.638,-88.074,169.558,38.784,157.293
C04392=1039.401,62.388,-88.056,169.556,38.783,157.293
C04393=1039.394,62.140,-88.039,169.554,38.782,157.293
C04394=1039.388,61.890,-88.021,169.552,38.783,157.293
C04395=1039.381,61.641,-88.004,169.550,38.782,157.293
C04396=1039.376,61.392,-87.986,169.548,38.782,157.293
C04397=1039.368,61.105,-87.966,169.546,38.781,157.293
C04398=1039.360,60.819,-87.946,169.544,38.781,157.292
C04399=1039.353,60.533,-87.926,169.542,38.780,157.292
C04400=1039.346,60.246,-87.906,169.539,38.779,157.292
C04401=1039.340,59.997,-87.888,169.537,38.779,157.292
C04402=1039.333,59.748,-87.871,169.535,38.778,157.292
C04403=1039.326,59.498,-87.853,169.533,38.779,157.292
C04404=1039.321,59.249,-87.836,169.531,38.778,157.292
C04405=1039.314,59.000,-87.819,169.529,38.778,157.291
C04406=1039.307,58.750,-87.801,169.527,38.777,157.291
C04407=1039.302,58.501,-87.784,169.525,38.776,157.291
C04408=1039.295,58.252,-87.766,169.523,38.776,157.291
C04409=1039.289,58.002,-87.748,169.521,38.775,157.291
C04410=1039.282,57.753,-87.731,169.519,38.776,157.291
C04411=1039.275,57.504,-87.714,169.517,38.775,157.291
C04412=1039.269,57.254,-87.696,169.515,38.774,157.291
C04413=1039.263,57.005,-87.679,169.513,38.774,157.290
C04414=1039.256,56.756,-87.662,169.511,38.773,157.290
C04415=1039.250,56.506,-87.644,169.509,38.773,157.290
C04416=1039.244,56.258,-87.627,169.507,38.772,157.290
C04417=1039.238,56.008,-87.609,169.505,38.772,157.290
C04418=1039.231,55.758,-87.592,169.503,38.772,157.290
C04419=1039.225,55.510,-87.575,169.501,38.771,157.290
C04420=1039.219,55.260,-87.557,169.499,38.771,157.289
C04421=1039.212,55.011,-87.540,169.497,38.770,157.289
C04422=1039.205,54.762,-87.522,169.495,38.770,157.289
C04423=1039.199,54.512,-87.504,169.493,38.769,157.289
C04424=1039.193,54.263,-87.487,169.491,38.769,157.289
C04425=1039.186,54.014,-87.470,169.489,38.768,157.289
C04426=1039.181,53.764,-87.453,169.487,38.768,157.289
C04427=1039.174,53.515,-87.436,169.485,38.768,157.289
C04428=1039.168,53.265,-87.418,169.483,38.767,157.288
C04429=1039.162,53.016,-87.401,169.481,38.767,157.288
C04430=1039.155,52.767,-87.384,169.479,38.766,157.288
C04431=1039.149,52.518,-87.366,169.477,38.766,157.288
C04432=1039.142,52.268,-87.349,169.475,38.765,157.288
C04433=1039.137,52.019,-87.333,169.473,38.765,157.288
C04434=1039.130,51.769,-87.315,169.470,38.764,157.287
C04435=1039.124,51.521,-87.298,169.469,38.764,157.287
C04436=1039.117,51.271,-87.280,169.467,38.763,157.287
C04437=1039.111,51.021,-87.262,169.465,38.763,157.287
C04438=1039.105,50.773,-87.245,169.463,38.763,157.287
C04439=1039.098,50.523,-87.229,169.461,38.762,157.287
C04440=1039.093,50.274,-87.211,169.459,38.762,157.287
C04441=1039.086,50.024,-87.194,169.457,38.761,157.287
C04442=1039.080,49.775,-87.177,169.455,38.761,157.286
C04443=1039.074,49.525,-87.160,169.452,38.760,157.286
C04444=1039.068,49.276,-87.143,169.451,38.759,157.286
C04445=1039.061,49.027,-87.125,169.449,38.759,157.286
C04446=1039.055,48.778,-87.108,169.447,38.758,157.286
C04447=1039.049,48.528,-87.091,169.445,38.758,157.286
C04448=1039.042,48.279,-87.074,169.443,38.757,157.285
C04449=1039.036,48.029,-87.056,169.441,38.757,157.285
C04450=1039.030,47.781,-87.039,169.439,38.756,157.285
C04451=1039.024,47.531,-87.023,169.436,38.756,157.285
C04452=1039.017,47.282,-87.006,169.434,38.755,157.285
C04453=1039.012,47.033,-86.988,169.433,38.755,157.285
C04454=1039.005,46.783,-86.972,169.431,38.755,157.285
C04455=1038.999,46.534,-86.955,169.429,38.754,157.285
C04456=1038.993,46.284,-86.937,169.427,38.754,157.284
C04457=1038.987,46.035,-86.920,169.425,38.753,157.284
C04458=1038.980,45.786,-86.903,169.423,38.753,157.284
C04459=1038.974,45.536,-86.885,169.421,38.752,157.284
C04460=1038.969,45.287,-86.869,169.418,38.752,157.284
C04461=1038.961,45.001,-86.849,169.416,38.751,157.284
C04462=1038.954,44.714,-86.830,169.414,38.751,157.284
C04463=1038.947,44.427,-86.810,169.412,38.750,157.283
C04464=1038.939,44.141,-86.791,169.410,38.749,157.283
C04465=1038.934,43.891,-86.774,169.408,38.748,157.283
C04466=1038.927,43.642,-86.756,169.406,38.748,157.283
C04467=1038.921,43.393,-86.740,169.403,38.747,157.283
C04468=1038.915,43.143,-86.722,169.401,38.747,157.283
C04469=1038.909,42.894,-86.705,169.399,38.747,157.282
C04470=1038.903,42.645,-86.689,169.397,38.746,157.282
C04471=1038.896,42.395,-86.672,169.395,38.746,157.282
C04472=1038.890,42.146,-86.655,169.394,38.745,157.282
C04473=1038.883,41.897,-86.638,169.392,38.745,157.282
C04474=1038.877,41.647,-86.622,169.390,38.745,157.282
C04475=1038.871,41.398,-86.605,169.388,38.744,157.282
C04476=1038.865,41.148,-86.588,169.385,38.744,157.282
C04477=1038.859,40.899,-86.572,169.383,38.743,157.281
C04478=1038.852,40.650,-86.555,169.381,38.743,157.281
C04479=1038.846,40.400,-86.538,169.379,38.742,157.281
C04480=1038.839,40.151,-86.521,169.377,38.742,157.281
C04481=1038.833,39.902,-86.505,169.375,38.742,157.281
C04482=1038.827,39.653,-86.488,169.373,38.741,157.281
C04483=1038.820,39.403,-86.471,169.371,38.741,157.281
C04484=1038.814,39.153,-86.455,169.370,38.740,157.280
C04485=1038.808,38.905,-86.438,169.367,38.740,157.280
C04486=1038.801,38.655,-86.421,169.365,38.739,157.280
C04487=1038.795,38.406,-86.404,169.363,38.739,157.280
C04488=1038.789,38.157,-86.388,169.361,38.739,157.280
C04489=1038.783,37.907,-86.372,169.359,38.738,157.280
C04490=1038.776,37.658,-86.355,169.357,38.738,157.280
C04491=1038.770,37.408,-86.338,169.355,38.737,157.280
C04492=1038.764,37.158,-86.322,169.353,38.737,157.279
C04493=1038.758,36.910,-86.305,169.351,38.737,157.279
C04494=1038.751,36.660,-86.288,169.348,38.736,157.279
C04495=1038.745,36.410,-86.272,169.346,38.736,157.279
C04496=1038.738,36.161,-86.256,169.344,38.735,157.279
C04497=1038.732,35.912,-86.239,169.342,38.735,157.279
C04498=1038.726,35.662,-86.223,169.340,38.735,157.279
C04499=1038.720,35.413,-86.206,169.339,38.734,157.279
C04500=1038.713,35.163,-86.190,169.337,38.734,157.278
C04501=1038.706,34.915,-86.173,169.335,38.734,157.278
C04502=1038.700,34.665,-86.157,169.333,38.733,157.278
C04503=1038.694,34.415,-86.140,169.331,38.733,157.278
C04504=1038.688,34.166,-86.124,169.328,38.732,157.278
C04505=1038.681,33.917,-86.107,169.326,38.732,157.278
C04506=1038.674,33.667,-86.091,169.324,38.732,157.278
C04507=1038.668,33.418,-86.075,169.322,38.731,157.278
C04508=1038.662,33.169,-86.059,169.320,38.731,157.277
C04509=1038.656,32.919,-86.042,169.318,38.731,157.277
C04510=1038.650,32.669,-86.026,169.316,38.730,157.277
C04511=1038.643,32.421,-86.009,169.314,38.730,157.277
C04512=1038.637,32.172,-85.993,169.312,38.729,157.277
C04513=1038.630,31.922,-85.977,169.310,38.729,157.277
C04514=1038.624,31.672,-85.960,169.308,38.729,157.277
C04515=1038.618,31.423,-85.944,169.305,38.728,157.277
C04516=1038.612,31.174,-85.928,169.303,38.728,157.276
C04517=1038.605,30.924,-85.912,169.301,38.728,157.276
C04518=1038.599,30.675,-85.895,169.299,38.727,157.276
C04519=1038.593,30.426,-85.879,169.297,38.727,157.276
C04520=1038.586,30.177,-85.863,169.295,38.726,157.276
C04521=1038.580,29.927,-85.846,169.294,38.726,157.276
C04522=1038.574,29.677,-85.830,169.292,38.726,157.276
C04523=1038.568,29.428,-85.814,169.290,38.725,157.276
C04524=1038.561,29.179,-85.798,169.287,38.725,157.276
C04525=1038.554,28.892,-85.778,169.284,38.724,157.275
C04526=1038.547,28.605,-85.761,169.282,38.724,157.275
C04527=1038.539,28.318,-85.742,169.280,38.723,157.275
C04528=1038.532,28.032,-85.723,169.278,38.723,157.275
C04529=1038.526,27.783,-85.707,169.276,38.723,157.275
C04530=1038.519,27.533,-85.690,169.274,38.722,157.275
C04531=1038.513,27.284,-85.675,169.272,38.722,157.275
C04532=1038.507,27.034,-85.658,169.270,38.722,157.275
C04533=1038.500,26.785,-85.643,169.268,38.721,157.274
C04534=1038.494,26.535,-85.627,169.265,38.721,157.274
C04535=1038.488,26.285,-85.611,169.263,38.721,157.274
C04536=1038.481,26.036,-85.595,169.261,38.720,157.274
C04537=1038.475,25.787,-85.579,169.259,38.720,157.274
C04538=1038.469,25.538,-85.563,169.257,38.720,157.274
C04539=1038.462,25.288,-85.546,169.255,38.720,157.274
C04540=1038.455,25.039,-85.531,169.253,38.719,157.274
C04541=1038.449,24.790,-85.515,169.251,38.719,157.274
C04542=1038.443,24.540,-85.498,169.249,38.719,157.273
C04543=1038.437,24.291,-85.483,169.247,38.718,157.273
C04544=1038.431,24.041,-85.467,169.244,38.718,157.273
C04545=1038.424,23.791,-85.451,169.242,38.718,157.273
C04546=1038.418,23.542,-85.435,169.240,38.717,157.273
C04547=1038.411,23.293,-85.419,169.238,38.717,157.273
C04548=1038.405,23.044,-85.403,169.236,38.717,157.273
C04549=1038.399,22.795,-85.387,169.234,38.716,157.273
C04550=1038.393,22.545,-85.371,169.232,38.716,157.272
C04551=1038.386,22.295,-85.356,169.230,38.716,157.272
C04552=1038.380,22.046,-85.339,169.228,38.715,157.272
C04553=1038.373,21.797,-85.324,169.226,38.715,157.272
C04554=1038.367,21.547,-85.307,169.224,38.715,157.272
C04555=1038.360,21.298,-85.292,169.222,38.714,157.272
C04556=1038.355,21.048,-85.276,169.219,38.714,157.272
C04557=1038.348,20.799,-85.261,169.217,38.713,157.272
C04558=1038.342,20.550,-85.244,169.215,38.713,157.272
C04559=1038.336,20.300,-85.228,169.213,38.713,157.271
C04560=1038.329,20.050,-85.213,169.211,38.712,157.271
C04561=1038.323,19.801,-85.196,169.209,38.712,157.271
C04562=1038.316,19.552,-85.181,169.207,38.712,157.271
C04563=1038.310,19.302,-85.166,169.205,38.711,157.271
C04564=1038.304,19.053,-85.150,169.203,38.711,157.271
C04565=1038.297,18.804,-85.134,169.201,38.711,157.271
C04566=1038.291,18.554,-85.119,169.198,38.710,157.271
C04567=1038.285,18.305,-85.103,169.196,38.711,157.271
C04568=1038.278,18.056,-85.087,169.194,38.710,157.270
C04569=1038.273,17.806,-85.072,169.192,38.709,157.270
C04570=1038.265,17.556,-85.056,169.190,38.710,157.270
C04571=1038.259,17.307,-85.040,169.188,38.709,157.270
C04572=1038.253,17.057,-85.024,169.186,38.709,157.270
C04573=1038.246,16.808,-85.009,169.184,38.709,157.270
C04574=1038.240,16.559,-84.993,169.182,38.708,157.270
C04575=1038.234,16.309,-84.977,169.180,38.708,157.270
C04576=1038.227,16.060,-84.962,169.178,38.708,157.270
C04577=1038.222,15.810,-84.946,169.176,38.707,157.269
C04578=1038.215,15.561,-84.931,169.174,38.707,157.269
C04579=1038.208,15.312,-84.915,169.171,38.707,157.269
C04580=1038.203,15.062,-84.899,169.168,38.706,157.269
C04581=1038.196,14.813,-84.884,169.166,38.706,157.269
C04582=1038.190,14.563,-84.869,169.164,38.706,157.269
C04583=1038.184,14.314,-84.853,169.162,38.705,157.269
C04584=1038.177,14.064,-84.838,169.160,38.705,157.269
C04585=1038.171,13.815,-84.822,169.158,38.705,157.269
C04586=1038.164,13.565,-84.807,169.156,38.705,157.269
C04587=1038.158,13.316,-84.791,169.154,38.705,157.268
C04588=1038.152,13.066,-84.776,169.152,38.705,157.268
C04589=1038.144,12.781,-84.758,169.150,38.704,157.268
C04590=1038.137,12.496,-84.740,169.146,38.704,157.268
C04591=1038.130,12.210,-84.723,169.144,38.704,157.268
C04592=1038.122,11.925,-84.706,169.142,38.703,157.268
C04593=1038.115,11.676,-84.690,169.140,38.703,157.268
C04594=1038.109,11.426,-84.675,169.137,38.703,157.268
C04595=1038.103,11.177,-84.660,169.135,38.703,157.268
C04596=1038.096,10.928,-84.645,169.133,38.702,157.268
C04597=1038.090,10.678,-84.630,169.131,38.703,157.268
C04598=1038.084,10.429,-84.613,169.129,38.702,157.267
C04599=1038.077,10.179,-84.598,169.127,38.702,157.267
C04600=1038.071,9.929,-84.583,169.125,38.702,157.267
C04601=1038.064,9.680,-84.568,169.123,38.702,157.267
C04602=1038.058,9.431,-84.553,169.121,38.701,157.267
C04603=1038.051,9.181,-84.538,169.118,38.701,157.267
C04604=1038.045,8.932,-84.522,169.116,38.701,157.267
C04605=1038.038,8.682,-84.507,169.114,38.700,157.267
C04606=1038.032,8.433,-84.492,169.112,38.700,157.267
C04607=1038.025,8.183,-84.477,169.109,38.700,157.267
C04608=1038.019,7.934,-84.462,169.107,38.700,157.266
C04609=1038.013,7.684,-84.447,169.105,38.699,157.266
C04610=1038.007,7.434,-84.431,169.103,38.700,157.266
C04611=1038.000,7.185,-84.416,169.101,38.699,157.266
C04612=1037.994,6.936,-84.401,169.099,38.699,157.266
C04613=1037.988,6.687,-84.386,169.097,38.699,157.266
C04614=1037.982,6.437,-84.371,169.095,38.699,157.266
C04615=1037.975,6.188,-84.355,169.093,38.698,157.266
C04616=1037.969,5.938,-84.341,169.091,38.698,157.266
C04617=1037.962,5.689,-84.326,169.088,38.698,157.266
C04618=1037.956,5.439,-84.311,169.086,38.697,157.265
C04619=1037.949,5.190,-84.295,169.083,38.697,157.265
C04620=1037.943,4.940,-84.280,169.081,38.697,157.265
C04621=1037.936,4.691,-84.265,169.079,38.697,157.265
C04622=1037.931,4.442,-84.250,169.077,38.696,157.265
C04623=1037.924,4.192,-84.236,169.075,38.697,157.265
C04624=1037.917,3.943,-84.220,169.073,38.696,157.265
C04625=1037.912,3.693,-84.204,169.071,38.696,157.265
C04626=1037.905,3.443,-84.189,169.069,38.696,157.265
C04627=1037.899,3.194,-84.174,169.067,38.695,157.265
C04628=1037.893,2.944,-84.160,169.065,38.695,157.265
C04629=1037.887,2.695,-84.145,169.062,38.695,157.264
C04630=1037.881,2.445,-84.130,169.059,38.695,157.264
C04631=1037.874,2.196,-84.114,169.057,38.694,157.264
C04632=1037.867,1.947,-84.099,169.055,38.694,157.264
C04633=1037.861,1.697,-84.084,169.053,38.694,157.264
C04634=1037.855,1.447,-84.069,169.051,38.694,157.264
C04635=1037.849,1.198,-84.055,169.049,38.693,157.264
C04636=1037.843,0.949,-84.040,169.047,38.693,157.264
C04637=1037.836,0.699,-84.025,169.045,38.693,157.264
C04638=1037.830,0.449,-84.010,169.043,38.693,157.264
C04639=1037.824,0.200,-83.995,169.041,38.693,157.264
C04640=1037.818,-0.049,-83.981,169.038,38.692,157.263
C04641=1037.811,-0.299,-83.966,169.036,38.692,157.263
C04642=1037.805,-0.549,-83.951,169.033,38.692,157.263
C04643=1037.798,-0.798,-83.936,169.031,38.691,157.263
C04644=1037.793,-1.047,-83.921,169.029,38.691,157.263
C04645=1037.786,-1.297,-83.906,169.027,38.691,157.263
C04646=1037.780,-1.546,-83.891,169.025,38.691,157.263
C04647=1037.773,-1.796,-83.876,169.023,38.690,157.263
C04648=1037.768,-2.045,-83.862,169.021,38.690,157.263
C04649=1037.761,-2.295,-83.847,169.019,38.690,157.262
C04650=1037.755,-2.544,-83.832,169.016,38.689,157.262
C04651=1037.749,-2.794,-83.817,169.014,38.690,157.262
C04652=1037.743,-3.043,-83.802,169.012,38.689,157.262
C04653=1037.736,-3.326,-83.785,169.010,38.689,157.262
C04654=1037.728,-3.610,-83.768,169.007,38.689,157.262
C04655=1037.721,-3.894,-83.752,169.004,38.688,157.262
C04656=1037.714,-4.177,-83.735,169.001,38.688,157.262
C04657=1037.708,-4.427,-83.720,168.999,38.688,157.262
C04658=1037.701,-4.676,-83.706,168.997,38.688,157.262
C04659=1037.695,-4.925,-83.691,168.995,38.688,157.262
C04660=1037.689,-5.175,-83.676,168.993,38.687,157.261
C04661=1037.682,-5.424,-83.662,168.991,38.688,157.261
C04662=1037.676,-5.674,-83.648,168.988,38.688,157.261
C04663=1037.670,-5.923,-83.633,168.986,38.687,157.261
C04664=1037.663,-6.173,-83.618,168.984,38.687,157.261
C04665=1037.656,-6.422,-83.604,168.982,38.687,157.261
C04666=1037.650,-6.671,-83.589,168.980,38.687,157.261
C04667=1037.644,-6.922,-83.575,168.978,38.687,157.261
C04668=1037.637,-7.171,-83.561,168.975,38.687,157.261
C04669=1037.631,-7.421,-83.546,168.973,38.687,157.261
C04670=1037.625,-7.670,-83.531,168.971,38.687,157.261
C04671=1037.618,-7.920,-83.518,168.968,38.686,157.261
C04672=1037.612,-8.169,-83.503,168.966,38.686,157.261
C04673=1037.606,-8.418,-83.488,168.964,38.686,157.260
C04674=1037.599,-8.668,-83.474,168.961,38.686,157.260
C04675=1037.593,-8.918,-83.459,168.959,38.686,157.260
C04676=1037.587,-9.167,-83.445,168.957,38.686,157.260
C04677=1037.580,-9.416,-83.431,168.955,38.686,157.260
C04678=1037.574,-9.666,-83.416,168.953,38.685,157.260
C04679=1037.568,-9.915,-83.402,168.950,38.685,157.260
C04680=1037.561,-10.165,-83.387,168.948,38.685,157.260
C04681=1037.555,-10.415,-83.373,168.946,38.685,157.260
C04682=1037.549,-10.664,-83.359,168.944,38.685,157.260
C04683=1037.542,-10.913,-83.344,168.942,38.684,157.260
C04684=1037.536,-11.163,-83.330,168.940,38.685,157.260
C04685=1037.530,-11.413,-83.315,168.937,38.685,157.260
C04686=1037.523,-11.663,-83.302,168.935,38.684,157.259
C04687=1037.518,-11.911,-83.287,168.933,38.684,157.259
C04688=1037.511,-12.161,-83.272,168.930,38.684,157.259
C04689=1037.505,-12.410,-83.259,168.928,38.684,157.259
C04690=1037.499,-12.660,-83.244,168.925,38.684,157.259
C04691=1037.492,-12.910,-83.230,168.923,38.684,157.259
C04692=1037.486,-13.159,-83.216,168.921,38.684,157.259
C04693=1037.480,-13.409,-83.201,168.919,38.683,157.259
C04694=1037.473,-13.658,-83.188,168.917,38.683,157.259
C04695=1037.467,-13.908,-83.173,168.914,38.683,157.259
C04696=1037.461,-14.158,-83.158,168.912,38.683,157.259
C04697=1037.454,-14.406,-83.144,168.910,38.683,157.259
C04698=1037.448,-14.657,-83.130,168.908,38.682,157.258
C04699=1037.442,-14.906,-83.116,168.906,38.683,157.258
C04700=1037.436,-15.156,-83.102,168.903,38.683,157.258
C04701=1037.430,-15.405,-83.087,168.901,38.682,157.258
C04702=1037.423,-15.655,-83.074,168.899,38.682,157.258
C04703=1037.417,-15.904,-83.059,168.897,38.682,157.258
C04704=1037.410,-16.154,-83.046,168.894,38.682,157.258
C04705=1037.403,-16.403,-83.031,168.891,38.682,157.258
C04706=1037.398,-16.652,-83.017,168.889,38.682,157.258
C04707=1037.391,-16.902,-83.004,168.887,38.682,157.258
C04708=1037.385,-17.151,-82.989,168.885,38.682,157.258
C04709=1037.378,-17.401,-82.976,168.882,38.682,157.258
C04710=1037.372,-17.650,-82.962,168.880,38.682,157.258
C04711=1037.366,-17.900,-82.947,168.878,38.682,157.258
C04712=1037.360,-18.150,-82.934,168.876,38.682,157.257
C04713=1037.353,-18.399,-82.920,168.873,38.682,157.257
C04714=1037.347,-18.648,-82.906,168.871,38.682,157.257
C04715=1037.340,-18.898,-82.892,168.869,38.682,157.257
C04716=1037.334,-19.148,-82.877,168.867,38.681,157.257
C04717=1037.327,-19.430,-82.862,168.864,38.682,157.257
C04718=1037.320,-19.712,-82.846,168.862,38.682,157.257
C04719=1037.313,-19.993,-82.831,168.859,38.681,157.257
C04720=1037.306,-20.275,-82.815,168.856,38.681,157.257
C04721=1037.299,-20.525,-82.801,168.854,38.682,157.257
C04722=1037.292,-20.774,-82.787,168.852,38.682,157.257
C04723=1037.286,-21.024,-82.773,168.850,38.681,157.257
C04724=1037.280,-21.273,-82.760,168.847,38.681,157.257
C04725=1037.274,-21.523,-82.746,168.845,38.681,157.257
C04726=1037.267,-21.772,-82.732,168.843,38.682,157.257
C04727=1037.261,-22.021,-82.718,168.840,38.681,157.256
C04728=1037.255,-22.272,-82.704,168.837,38.681,157.256
C04729=1037.249,-22.521,-82.691,168.835,38.681,157.256
C04730=1037.242,-22.770,-82.677,168.833,38.681,157.256
C04731=1037.236,-23.020,-82.663,168.831,38.681,157.256
C04732=1037.229,-23.270,-82.649,168.828,38.681,157.256
C04733=1037.223,-23.519,-82.636,168.826,38.681,157.256
C04734=1037.218,-23.769,-82.622,168.824,38.681,157.256
C04735=1037.211,-24.018,-82.608,168.821,38.681,157.256
C04736=1037.204,-24.267,-82.594,168.819,38.681,157.256
C04737=1037.198,-24.518,-82.580,168.817,38.681,157.256
C04738=1037.192,-24.767,-82.567,168.815,38.680,157.256
C04739=1037.186,-25.016,-82.553,168.812,38.681,157.256
C04740=1037.180,-25.266,-82.539,168.810,38.681,157.256
C04741=1037.174,-25.516,-82.526,168.808,38.681,157.256
C04742=1037.167,-25.764,-82.512,168.806,38.680,157.256
C04743=1037.161,-26.015,-82.498,168.803,38.680,157.255
C04744=1037.155,-26.264,-82.484,168.801,38.681,157.255
C04745=1037.148,-26.514,-82.471,168.799,38.680,157.255
C04746=1037.143,-26.763,-82.457,168.796,38.680,157.255
C04747=1037.136,-27.013,-82.444,168.794,38.680,157.255
C04748=1037.129,-27.263,-82.430,168.792,38.680,157.255
C04749=1037.123,-27.512,-82.417,168.790,38.681,157.255
C04750=1037.116,-27.762,-82.403,168.786,38.681,157.255
C04751=1037.111,-28.011,-82.389,168.784,38.680,157.255
C04752=1037.105,-28.261,-82.376,168.782,38.680,157.255
C04753=1037.098,-28.511,-82.362,168.779,38.680,157.255
C04754=1037.092,-28.760,-82.349,168.777,38.681,157.255
C04755=1037.086,-29.009,-82.336,168.775,38.681,157.255
C04756=1037.079,-29.259,-82.322,168.772,38.681,157.255
C04757=1037.072,-29.508,-82.309,168.770,38.681,157.255
C04758=1037.066,-29.758,-82.296,168.768,38.681,157.255
C04759=1037.059,-30.008,-82.282,168.765,38.681,157.255
C04760=1037.053,-30.257,-82.269,168.763,38.681,157.255
C04761=1037.047,-30.506,-82.256,168.761,38.681,157.255
C04762=1037.040,-30.756,-82.242,168.758,38.681,157.254
C04763=1037.034,-31.006,-82.229,168.756,38.681,157.254
C04764=1037.028,-31.255,-82.216,168.754,38.681,157.254
C04765=1037.022,-31.506,-82.202,168.751,38.681,157.254
C04766=1037.016,-31.755,-82.189,168.749,38.682,157.254
C04767=1037.010,-32.004,-82.175,168.747,38.682,157.254
C04768=1037.003,-32.253,-82.162,168.744,38.682,157.254
C04769=1036.997,-32.503,-82.148,168.742,38.681,157.254
C04770=1036.990,-32.753,-82.135,168.740,38.681,157.254
C04771=1036.984,-33.003,-82.123,168.737,38.682,157.254
C04772=1036.978,-33.252,-82.109,168.735,38.682,157.254
C04773=1036.971,-33.502,-82.096,168.733,38.682,157.254
C04774=1036.965,-33.751,-82.082,168.730,38.682,157.254
C04775=1036.959,-34.000,-82.069,168.728,38.682,157.254
C04776=1036.952,-34.251,-82.056,168.726,38.682,157.254
C04777=1036.946,-34.500,-82.043,168.723,38.682,157.254
C04778=1036.940,-34.749,-82.030,168.721,38.682,157.254
C04779=1036.934,-34.999,-82.016,168.719,38.682,157.254
C04780=1036.928,-35.248,-82.003,168.716,38.682,157.254
C04781=1036.921,-35.530,-81.988,168.714,38.682,157.254
C04782=1036.914,-35.811,-81.974,168.710,38.682,157.254
C04783=1036.906,-36.092,-81.959,168.707,38.683,157.254
C04784=1036.900,-36.373,-81.944,168.705,38.683,157.253
C04785=1036.893,-36.623,-81.930,168.702,38.683,157.253
C04786=1036.887,-36.872,-81.917,168.700,38.683,157.253
C04787=1036.881,-37.122,-81.904,168.697,38.682,157.253
C04788=1036.875,-37.371,-81.891,168.695,38.683,157.253
C04789=1036.869,-37.621,-81.878,168.693,38.683,157.253
C04790=1036.863,-37.870,-81.865,168.690,38.683,157.253
C04791=1036.856,-38.120,-81.852,168.688,38.683,157.253
C04792=1036.850,-38.370,-81.838,168.686,38.683,157.253
C04793=1036.844,-38.620,-81.826,168.683,38.683,157.253
C04794=1036.838,-38.869,-81.813,168.681,38.683,157.253
C04795=1036.831,-39.118,-81.799,168.679,38.683,157.253
C04796=1036.825,-39.368,-81.787,168.676,38.684,157.253
C04797=1036.818,-39.618,-81.774,168.674,38.684,157.253
C04798=1036.812,-39.867,-81.761,168.671,38.684,157.253
C04799=1036.806,-40.117,-81.748,168.669,38.684,157.253
C04800=1036.800,-40.367,-81.735,168.667,38.684,157.253
C04801=1036.793,-40.616,-81.723,168.664,38.684,157.253
C04802=1036.787,-40.865,-81.710,168.662,38.684,157.253
C04803=1036.780,-41.115,-81.696,168.659,38.685,157.253
C04804=1036.774,-41.365,-81.684,168.657,38.685,157.253
C04805=1036.767,-41.614,-81.671,168.654,38.685,157.253
C04806=1036.761,-41.864,-81.659,168.652,38.685,157.253
C04807=1036.755,-42.113,-81.645,168.650,38.685,157.253
C04808=1036.749,-42.363,-81.633,168.647,38.685,157.253
C04809=1036.743,-42.613,-81.620,168.645,38.685,157.253
C04810=1036.736,-42.862,-81.608,168.642,38.686,157.252
C04811=1036.730,-43.111,-81.594,168.640,38.686,157.253
C04812=1036.724,-43.362,-81.581,168.638,38.686,157.253
C04813=1036.717,-43.611,-81.568,168.635,38.687,157.252
C04814=1036.711,-43.861,-81.556,168.633,38.687,157.252
C04815=1036.705,-44.110,-81.543,168.630,38.687,157.252
C04816=1036.699,-44.360,-81.530,168.628,38.687,157.252
C04817=1036.693,-44.610,-81.518,168.625,38.687,157.252
C04818=1036.686,-44.859,-81.505,168.623,38.687,157.252
C04819=1036.680,-45.109,-81.493,168.621,38.687,157.252
C04820=1036.674,-45.358,-81.479,168.618,38.688,157.252
C04821=1036.667,-45.607,-81.467,168.616,38.688,157.252
C04822=1036.661,-45.857,-81.455,168.613,38.688,157.252
C04823=1036.655,-46.107,-81.442,168.611,38.688,157.252
C04824=1036.649,-46.357,-81.429,168.608,38.688,157.252
C04825=1036.642,-46.606,-81.417,168.606,38.688,157.252
C04826=1036.636,-46.855,-81.404,168.604,38.688,157.252
C04827=1036.630,-47.105,-81.391,168.601,38.689,157.252
C04828=1036.624,-47.355,-81.379,168.599,38.689,157.252
C04829=1036.617,-47.604,-81.366,168.596,38.689,157.252
C04830=1036.611,-47.854,-81.353,168.594,38.690,157.252
C04831=1036.606,-48.104,-81.341,168.591,38.690,157.252
C04832=1036.599,-48.353,-81.328,168.589,38.690,157.252
C04833=1036.593,-48.603,-81.316,168.587,38.690,157.252
C04834=1036.587,-48.853,-81.303,168.584,38.690,157.252
C04835=1036.581,-49.102,-81.291,168.582,38.690,157.252
C04836=1036.574,-49.351,-81.278,168.579,38.690,157.252
C04837=1036.568,-49.601,-81.265,168.577,38.691,157.252
C04838=1036.562,-49.851,-81.253,168.574,38.691,157.252
C04839=1036.555,-50.101,-81.241,168.572,38.691,157.252
C04840=1036.549,-50.350,-81.228,168.569,38.691,157.252
C04841=1036.543,-50.600,-81.215,168.567,38.691,157.252
C04842=1036.537,-50.849,-81.203,168.565,38.692,157.252
C04843=1036.531,-51.099,-81.190,168.562,38.692,157.252
C04844=1036.524,-51.349,-81.179,168.560,38.692,157.252
C04845=1036.517,-51.630,-81.164,168.557,38.693,157.252
C04846=1036.510,-51.911,-81.151,168.554,38.693,157.252
C04847=1036.503,-52.193,-81.138,168.551,38.693,157.252
C04848=1036.495,-52.475,-81.123,168.548,38.694,157.252
C04849=1036.489,-52.724,-81.111,168.546,38.694,157.252
C04850=1036.483,-52.974,-81.099,168.543,38.694,157.252
C04851=1036.476,-53.224,-81.087,168.541,38.695,157.252
C04852=1036.469,-53.473,-81.075,168.538,38.695,157.252
C04853=1036.463,-53.723,-81.062,168.536,38.696,157.252
C04854=1036.457,-53.973,-81.050,168.533,38.696,157.252
C04855=1036.450,-54.222,-81.038,168.531,38.696,157.252
C04856=1036.445,-54.472,-81.026,168.528,38.697,157.252
C04857=1036.438,-54.721,-81.014,168.526,38.697,157.252
C04858=1036.432,-54.971,-81.002,168.523,38.698,157.252
C04859=1036.426,-55.221,-80.990,168.520,38.698,157.252
C04860=1036.419,-55.470,-80.978,168.518,38.699,157.252
C04861=1036.412,-55.720,-80.966,168.515,38.699,157.252
C04862=1036.406,-55.970,-80.953,168.513,38.699,157.252
C04863=1036.400,-56.219,-80.941,168.510,38.700,157.252
C04864=1036.393,-56.469,-80.929,168.508,38.700,157.252
C04865=1036.387,-56.719,-80.917,168.505,38.700,157.252
C04866=1036.381,-56.968,-80.905,168.503,38.701,157.252
C04867=1036.375,-57.217,-80.893,168.500,38.701,157.252
C04868=1036.369,-57.467,-80.881,168.498,38.701,157.252
C04869=1036.362,-57.717,-80.869,168.495,38.702,157.252
C04870=1036.356,-57.967,-80.857,168.493,38.702,157.252
C04871=1036.350,-58.217,-80.845,168.490,38.702,157.252
C04872=1036.344,-58.466,-80.833,168.488,38.703,157.252
C04873=1036.337,-58.715,-80.821,168.485,38.703,157.252
C04874=1036.331,-58.965,-80.809,168.483,38.703,157.252
C04875=1036.324,-59.215,-80.797,168.480,38.704,157.252
C04876=1036.318,-59.465,-80.786,168.477,38.704,157.252
C04877=1036.312,-59.714,-80.774,168.475,38.704,157.252
C04878=1036.306,-59.964,-80.761,168.472,38.705,157.252
C04879=1036.300,-60.213,-80.749,168.470,38.705,157.252
C04880=1036.293,-60.463,-80.737,168.467,38.705,157.252
C04881=1036.287,-60.713,-80.725,168.465,38.706,157.252
C04882=1036.281,-60.962,-80.714,168.462,38.706,157.252
C04883=1036.275,-61.212,-80.702,168.460,38.706,157.252
C04884=1036.268,-61.461,-80.690,168.457,38.707,157.252
C04885=1036.262,-61.711,-80.678,168.455,38.707,157.252
C04886=1036.256,-61.961,-80.666,168.452,38.708,157.252
C04887=1036.250,-62.210,-80.655,168.449,38.708,157.252
C04888=1036.244,-62.460,-80.642,168.447,38.709,157.252
C04889=1036.237,-62.710,-80.630,168.444,38.709,157.252
C04890=1036.231,-62.959,-80.619,168.442,38.709,157.252
C04891=1036.225,-63.209,-80.607,168.439,38.710,157.252
C04892=1036.219,-63.459,-80.595,168.437,38.710,157.252
C04893=1036.212,-63.709,-80.584,168.435,38.711,157.252
C04894=1036.206,-63.958,-80.572,168.433,38.711,157.252
C04895=1036.200,-64.207,-80.560,168.430,38.712,157.252
C04896=1036.194,-64.457,-80.547,168.428,38.712,157.252
C04897=1036.188,-64.707,-80.537,168.425,38.712,157.252
C04898=1036.181,-64.956,-80.525,168.422,38.713,157.252
C04899=1036.176,-65.206,-80.512,168.420,38.713,157.252
C04900=1036.170,-65.455,-80.501,168.417,38.713,157.252
C04901=1036.163,-65.705,-80.489,168.415,38.714,157.252
C04902=1036.157,-65.955,-80.478,168.412,38.714,157.252
C04903=1036.152,-66.204,-80.466,168.410,38.714,157.252
C04904=1036.145,-66.454,-80.454,168.407,38.715,157.252
C04905=1036.139,-66.704,-80.443,168.405,38.715,157.252
C04906=1036.133,-66.953,-80.431,168.402,38.716,157.252
C04907=1036.126,-67.203,-80.420,168.399,38.716,157.252
C04908=1036.120,-67.453,-80.407,168.397,38.716,157.252
C04909=1036.113,-67.748,-80.394,168.394,38.717,157.252
C04910=1036.106,-68.044,-80.380,168.391,38.717,157.252
C04911=1036.098,-68.339,-80.366,168.388,38.718,157.252
C04912=1036.091,-68.634,-80.353,168.385,38.718,157.252
C04913=1036.086,-68.885,-80.341,168.382,38.718,157.252
C04914=1036.079,-69.134,-80.329,168.380,38.719,157.252
C04915=1036.073,-69.384,-80.318,168.377,38.719,157.252
C04916=1036.067,-69.633,-80.306,168.374,38.720,157.252
C04917=1036.061,-69.883,-80.295,168.372,38.720,157.252
C04918=1036.055,-70.133,-80.282,168.369,38.720,157.252
C04919=1036.049,-70.382,-80.272,168.367,38.721,157.252
C04920=1036.043,-70.632,-80.260,168.364,38.721,157.252
C04921=1036.036,-70.882,-80.248,168.362,38.722,157.252
C04922=1036.030,-71.131,-80.237,168.359,38.722,157.252
C04923=1036.025,-71.381,-80.225,168.356,38.722,157.252
C04924=1036.019,-71.631,-80.214,168.354,38.723,157.252
C04925=1036.013,-71.874,-80.202,168.351,38.723,157.252
C04926=1036.006,-72.117,-80.191,168.349,38.723,157.252
C04927=1036.000,-72.361,-80.180,168.346,38.724,157.252
C04928=1035.995,-72.603,-80.169,168.344,38.724,157.252
C04929=1035.990,-72.847,-80.158,168.341,38.725,157.252
C04930=1035.984,-73.091,-80.147,168.339,38.725,157.252
C04931=1035.978,-73.334,-80.136,168.336,38.725,157.252
C04932=1035.972,-73.577,-80.125,168.334,38.726,157.252
C04933=1035.965,-73.827,-80.113,168.331,38.726,157.252
C04934=1035.959,-74.077,-80.102,168.328,38.727,157.252
C04935=1035.953,-74.326,-80.091,168.326,38.727,157.252
C04936=1035.947,-74.576,-80.079,168.324,38.728,157.252
C04937=1035.941,-74.825,-80.068,168.322,38.728,157.252
C04938=1035.935,-75.076,-80.057,168.319,38.729,157.252
C04939=1035.929,-75.325,-80.046,168.316,38.730,157.252
C04940=1035.922,-75.575,-80.034,168.314,38.730,157.252
C04941=1035.917,-75.824,-80.023,168.311,38.731,157.252
C04942=1035.910,-76.074,-80.012,168.308,38.731,157.252
C04943=1035.904,-76.324,-80.001,168.306,38.732,157.252
C04944=1035.898,-76.574,-79.990,168.303,38.733,157.252
C04945=1035.892,-76.823,-79.978,168.300,38.733,157.252
C04946=1035.886,-77.072,-79.967,168.298,38.734,157.252
C04947=1035.879,-77.322,-79.956,168.295,38.734,157.252
C04948=1035.874,-77.572,-79.946,168.293,38.735,157.252
C04949=1035.867,-77.822,-79.934,168.290,38.735,157.253
C04950=1035.861,-78.071,-79.923,168.287,38.736,157.252
C04951=1035.855,-78.321,-79.912,168.285,38.736,157.253
C04952=1035.849,-78.570,-79.901,168.282,38.737,157.253
C04953=1035.843,-78.821,-79.889,168.279,38.737,157.253
C04954=1035.837,-79.070,-79.879,168.277,38.738,157.253
C04955=1035.831,-79.320,-79.868,168.274,38.738,157.253
C04956=1035.825,-79.570,-79.856,168.271,38.739,157.253
C04957=1035.818,-79.819,-79.846,168.270,38.740,157.253
C04958=1035.812,-80.069,-79.835,168.267,38.740,157.253
C04959=1035.806,-80.319,-79.824,168.264,38.741,157.253
C04960=1035.800,-80.569,-79.813,168.262,38.742,157.253
C04961=1035.794,-80.818,-79.802,168.259,38.743,157.253
C04962=1035.788,-81.068,-79.792,168.256,38.743,157.253
C04963=1035.781,-81.318,-79.780,168.254,38.744,157.253
C04964=1035.775,-81.567,-79.770,168.251,38.744,157.253
C04965=1035.769,-81.817,-79.759,168.248,38.745,157.253
C04966=1035.763,-82.067,-79.748,168.246,38.746,157.253
C04967=1035.756,-82.316,-79.738,168.243,38.746,157.253
C04968=1035.750,-82.566,-79.726,168.240,38.747,157.253
C04969=1035.744,-82.815,-79.716,168.237,38.748,157.253
C04970=1035.737,-83.065,-79.705,168.235,38.749,157.253
C04971=1035.731,-83.315,-79.694,168.232,38.749,157.253
C04972=1035.725,-83.564,-79.684,168.229,38.750,157.253
C04973=1035.718,-83.849,-79.671,168.227,38.750,157.254
C04974=1035.711,-84.134,-79.659,168.224,38.751,157.254
C04975=1035.704,-84.419,-79.647,168.221,38.752,157.254
C04976=1035.697,-84.703,-79.635,168.218,38.753,157.254
C04977=1035.691,-84.954,-79.624,168.215,38.754,157.254
C04978=1035.685,-85.204,-79.613,168.213,38.755,157.254
C04979=1035.678,-85.453,-79.603,168.210,38.755,157.254
C04980=1035.672,-85.703,-79.592,168.207,38.756,157.254
C04981=1035.666,-85.953,-79.581,168.204,38.756,157.254
C04982=1035.660,-86.202,-79.570,168.202,38.757,157.254
C04983=1035.654,-86.453,-79.560,168.199,38.758,157.254
C04984=1035.647,-86.702,-79.550,168.196,38.759,157.254
C04985=1035.642,-86.951,-79.539,168.194,38.760,157.254
C04986=1035.636,-87.201,-79.528,168.191,38.760,157.254
C04987=1035.629,-87.451,-79.517,168.189,38.761,157.254
C04988=1035.623,-87.701,-79.507,168.186,38.762,157.254
C04989=1035.618,-87.950,-79.496,168.184,38.762,157.254
C04990=1035.610,-88.200,-79.486,168.181,38.763,157.255
C04991=1035.605,-88.450,-79.475,168.178,38.764,157.255
C04992=1035.599,-88.699,-79.465,168.176,38.765,157.255
///RCONF 1,0,0,0,1,0,0,0,0,0,0,0,0,0,0,0,0,0,0,0,0,0,0,0
C04993=1035.593,-88.949,-79.454,168.173,38.765,157.255
C04994=1035.587,-89.198,-79.443,168.170,38.766,157.255
C04995=1035.580,-89.448,-79.433,168.167,38.767,157.255
C04996=1035.575,-89.698,-79.423,168.165,38.767,157.255
C04997=1035.568,-89.947,-79.412,168.162,38.768,157.255
C04998=1035.562,-90.197,-79.401,168.159,38.769,157.255
C04999=1035.556,-90.447,-79.391,168.158,38.770,157.255
C05000=1035.550,-90.697,-79.381,168.154,38.770,157.255
C05001=1035.544,-90.946,-79.370,168.152,38.771,157.255
C05002=1035.538,-91.196,-79.360,168.149,38.772,157.255
C05003=1035.532,-91.446,-79.349,168.147,38.772,157.255
C05004=1035.525,-91.696,-79.339,168.144,38.773,157.255
C05005=1035.520,-91.946,-79.328,168.141,38.774,157.255
C05006=1035.514,-92.195,-79.318,168.139,38.775,157.256
C05007=1035.507,-92.444,-79.307,168.136,38.775,157.255
C05008=1035.502,-92.694,-79.297,168.133,38.776,157.256
C05009=1035.496,-92.944,-79.287,168.130,38.777,157.256
C05010=1035.490,-93.194,-79.277,168.128,38.778,157.256
C05011=1035.483,-93.444,-79.266,168.125,38.778,157.256
C05012=1035.477,-93.693,-79.255,168.122,38.779,157.256
C05013=1035.471,-93.943,-79.246,168.120,38.780,157.256
C05014=1035.465,-94.192,-79.235,168.118,38.781,157.256
C05015=1035.460,-94.443,-79.225,168.115,38.782,157.256
C05016=1035.453,-94.692,-79.214,168.112,38.782,157.256
C05017=1035.448,-94.942,-79.204,168.110,38.783,157.256
C05018=1035.442,-95.191,-79.194,168.107,38.784,157.256
C05019=1035.436,-95.441,-79.184,168.104,38.784,157.256
C05020=1035.429,-95.691,-79.173,168.101,38.785,157.256
C05021=1035.424,-95.941,-79.163,168.099,38.786,157.256
C05022=1035.417,-96.190,-79.153,168.096,38.787,157.256
C05023=1035.412,-96.440,-79.142,168.093,38.788,157.257
C05024=1035.406,-96.690,-79.132,168.090,38.789,157.257
C05025=1035.400,-96.940,-79.122,168.088,38.789,157.257
C05026=1035.394,-97.189,-79.111,168.085,38.789,157.257
C05027=1035.388,-97.439,-79.102,168.083,38.790,157.257
C05028=1035.382,-97.689,-79.091,168.080,38.791,157.257
C05029=1035.376,-97.938,-79.081,168.078,38.793,157.257
C05030=1035.370,-98.188,-79.071,168.075,38.793,157.257
C05031=1035.363,-98.437,-79.061,168.072,38.794,157.257
C05032=1035.358,-98.687,-79.051,168.069,38.795,157.257
C05033=1035.352,-98.937,-79.041,168.067,38.796,157.257
C05034=1035.345,-99.187,-79.031,168.064,38.797,157.257
C05035=1035.339,-99.437,-79.021,168.061,38.798,157.257
C05036=1035.333,-99.687,-79.011,168.058,38.798,157.257
C05037=1035.326,-99.974,-79.000,168.056,38.799,157.258
C05038=1035.319,-100.261,-78.988,168.053,38.801,157.258
C05039=1035.312,-100.548,-78.976,168.050,38.802,157.258
C05040=1035.305,-100.835,-78.965,168.046,38.803,157.258
C05041=1035.299,-101.085,-78.956,168.044,38.803,157.258
C05042=1035.293,-101.335,-78.945,168.041,38.805,157.258
C05043=1035.287,-101.584,-78.935,168.038,38.806,157.258
C05044=1035.281,-101.834,-78.926,168.035,38.807,157.258
C05045=1035.275,-102.084,-78.915,168.032,38.807,157.258
C05046=1035.269,-102.334,-78.906,168.031,38.808,157.258
C05047=1035.262,-102.583,-78.896,168.028,38.809,157.258
C05048=1035.256,-102.833,-78.886,168.025,38.810,157.259
C05049=1035.251,-103.083,-78.876,168.022,38.811,157.259
C05050=1035.245,-103.333,-78.866,168.020,38.812,157.259
C05051=1035.239,-103.582,-78.857,168.017,38.813,157.259
C05052=1035.233,-103.832,-78.848,168.014,38.814,157.259
C05053=1035.227,-104.081,-78.837,168.011,38.815,157.259
C05054=1035.221,-104.331,-78.827,168.008,38.816,157.259
C05055=1035.215,-104.581,-78.818,168.006,38.816,157.259
C05056=1035.209,-104.831,-78.808,168.004,38.818,157.259
C05057=1035.203,-105.080,-78.798,168.001,38.819,157.259
C05058=1035.197,-105.331,-78.788,167.998,38.820,157.260
C05059=1035.191,-105.580,-78.779,167.995,38.820,157.260
C05060=1035.185,-105.830,-78.769,167.993,38.821,157.260
C05061=1035.178,-106.079,-78.759,167.990,38.822,157.260
C05062=1035.172,-106.329,-78.749,167.987,38.823,157.260
C05063=1035.167,-106.579,-78.739,167.984,38.824,157.260
C05064=1035.161,-106.828,-78.730,167.981,38.825,157.260
C05065=1035.155,-107.078,-78.720,167.980,38.826,157.260
C05066=1035.149,-107.328,-78.711,167.977,38.827,157.260
C05067=1035.143,-107.578,-78.701,167.974,38.828,157.260
C05068=1035.136,-107.828,-78.692,167.971,38.829,157.260
C05069=1035.130,-108.077,-78.682,167.968,38.830,157.261
C05070=1035.124,-108.327,-78.673,167.965,38.832,157.261
C05071=1035.118,-108.577,-78.663,167.963,38.832,157.261
C05072=1035.113,-108.826,-78.653,167.960,38.833,157.261
C05073=1035.107,-109.076,-78.644,167.958,38.834,157.261
C05074=1035.101,-109.326,-78.634,167.955,38.836,157.261
C05075=1035.095,-109.576,-78.624,167.952,38.836,157.261
C05076=1035.088,-109.826,-78.615,167.949,38.837,157.261
C05077=1035.082,-110.075,-78.605,167.947,38.839,157.261
C05078=1035.076,-110.326,-78.596,167.944,38.840,157.262
C05079=1035.071,-110.575,-78.587,167.941,38.840,157.262
C05080=1035.065,-110.825,-78.578,167.938,38.842,157.262
C05081=1035.058,-111.074,-78.568,167.936,38.843,157.262
C05082=1035.052,-111.324,-78.559,167.933,38.844,157.262
C05083=1035.046,-111.574,-78.549,167.931,38.845,157.262
C05084=1035.041,-111.823,-78.540,167.928,38.846,157.262
C05085=1035.034,-112.073,-78.530,167.925,38.847,157.262
C05086=1035.029,-112.323,-78.521,167.922,38.848,157.262
C05087=1035.022,-112.573,-78.512,167.919,38.849,157.263
C05088=1035.016,-112.823,-78.502,167.916,38.850,157.263
C05089=1035.011,-113.072,-78.493,167.915,38.851,157.263
C05090=1035.004,-113.322,-78.483,167.912,38.852,157.263
C05091=1034.998,-113.572,-78.474,167.909,38.853,157.263
C05092=1034.992,-113.822,-78.465,167.906,38.855,157.263
C05093=1034.987,-114.071,-78.456,167.903,38.855,157.263
C05094=1034.981,-114.321,-78.446,167.900,38.857,157.263
C05095=1034.974,-114.571,-78.437,167.898,38.858,157.263
C05096=1034.969,-114.821,-78.428,167.895,38.859,157.263
C05097=1034.963,-115.070,-78.419,167.893,38.860,157.264
C05098=1034.957,-115.320,-78.409,167.890,38.861,157.264
C05099=1034.951,-115.570,-78.400,167.887,38.863,157.264
C05100=1034.945,-115.820,-78.391,167.884,38.863,157.264
C05101=1034.938,-116.106,-78.381,167.881,38.865,157.264
C05102=1034.931,-116.392,-78.370,167.878,38.866,157.264
C05103=1034.925,-116.679,-78.359,167.874,38.867,157.264
C05104=1034.917,-116.965,-78.349,167.872,38.869,157.265
C05105=1034.911,-117.216,-78.340,167.869,38.870,157.265
C05106=1034.906,-117.465,-78.331,167.866,38.871,157.265
C05107=1034.899,-117.715,-78.321,167.864,38.872,157.265
C05108=1034.894,-117.965,-78.312,167.861,38.874,157.265
C05109=1034.887,-118.215,-78.303,167.858,38.874,157.265
C05110=1034.881,-118.464,-78.295,167.856,38.876,157.265
C05111=1034.875,-118.714,-78.285,167.853,38.877,157.265
C05112=1034.869,-118.964,-78.276,167.850,38.878,157.266
C05113=1034.864,-119.214,-78.267,167.847,38.879,157.266
C05114=1034.858,-119.463,-78.258,167.844,38.881,157.266
C05115=1034.852,-119.713,-78.250,167.842,38.881,157.266
C05116=1034.846,-119.963,-78.240,167.839,38.883,157.266
C05117=1034.840,-120.213,-78.231,167.836,38.884,157.266
C05118=1034.834,-120.462,-78.222,167.834,38.885,157.266
C05119=1034.828,-120.712,-78.213,167.831,38.886,157.266
C05120=1034.822,-120.962,-78.204,167.828,38.888,157.267
C05121=1034.816,-121.211,-78.195,167.825,38.889,157.267
C05122=1034.810,-121.462,-78.186,167.822,38.890,157.267
C05123=1034.804,-121.711,-78.177,167.820,38.892,157.267
C05124=1034.798,-121.961,-78.168,167.818,38.892,157.267
C05125=1034.792,-122.211,-78.159,167.815,38.894,157.267
C05126=1034.786,-122.460,-78.151,167.812,38.895,157.267
C05127=1034.780,-122.711,-78.142,167.809,38.896,157.268
C05128=1034.775,-122.960,-78.133,167.806,38.897,157.268
C05129=1034.768,-123.210,-78.124,167.803,38.899,157.268
C05130=1034.763,-123.459,-78.115,167.800,38.900,157.268
C05131=1034.757,-123.709,-78.106,167.798,38.901,157.268
C05132=1034.751,-123.959,-78.097,167.796,38.903,157.268
C05133=1034.745,-124.209,-78.088,167.793,38.903,157.268
C05134=1034.739,-124.459,-78.080,167.790,38.905,157.268
C05135=1034.733,-124.708,-78.071,167.787,38.906,157.269
C05136=1034.727,-124.959,-78.062,167.784,38.907,157.269
C05137=1034.721,-125.208,-78.054,167.782,38.909,157.269
C05138=1034.715,-125.458,-78.045,167.779,38.910,157.269
C05139=1034.709,-125.707,-78.037,167.776,38.911,157.269
C05140=1034.703,-125.958,-78.028,167.773,38.913,157.269
C05141=1034.698,-126.207,-78.019,167.770,38.914,157.270
C05142=1034.691,-126.457,-78.010,167.768,38.915,157.270
C05143=1034.685,-126.707,-78.002,167.766,38.917,157.270
C05144=1034.680,-126.956,-77.992,167.763,38.918,157.270
C05145=1034.674,-127.206,-77.984,167.760,38.919,157.270
C05146=1034.668,-127.456,-77.976,167.757,38.920,157.270
C05147=1034.661,-127.705,-77.967,167.754,38.922,157.270
C05148=1034.656,-127.955,-77.958,167.751,38.923,157.270
C05149=1034.651,-128.205,-77.948,167.749,38.924,157.271
C05150=1034.646,-128.455,-77.939,167.746,38.924,157.270
C05151=1034.643,-128.704,-77.929,167.744,38.924,157.270
C05152=1034.640,-128.954,-77.918,167.742,38.923,157.270
C05153=1034.639,-129.203,-77.905,167.740,38.922,157.270
C05154=1034.637,-129.454,-77.893,167.738,38.920,157.270
C05155=1034.636,-129.704,-77.880,167.735,38.918,157.269
C05156=1034.635,-129.953,-77.867,167.734,38.916,157.269
C05157=1034.636,-130.203,-77.853,167.731,38.913,157.268
C05158=1034.638,-130.453,-77.838,167.730,38.910,157.268
C05159=1034.640,-130.703,-77.823,167.728,38.906,157.267
C05160=1034.643,-130.953,-77.807,167.727,38.901,157.266
C05161=1034.646,-131.203,-77.790,167.726,38.897,157.265
C05162=1034.650,-131.453,-77.773,167.725,38.891,157.264
C05163=1034.654,-131.704,-77.756,167.723,38.886,157.263
C05164=1034.660,-131.953,-77.737,167.722,38.879,157.262
C05165=1034.328,-131.978,-78.020,167.673,39.099,157.298
C05166=1034.322,-131.729,-78.039,167.674,39.106,157.299
C05167=1034.318,-131.478,-78.056,167.675,39.111,157.300
C05168=1034.314,-131.228,-78.074,167.677,39.117,157.301
C05169=1034.310,-130.978,-78.089,167.678,39.121,157.302
C05170=1034.307,-130.728,-78.106,167.680,39.126,157.302
C05171=1034.305,-130.479,-78.121,167.681,39.129,157.303
C05172=1034.304,-130.228,-78.136,167.683,39.133,157.304
C05173=1034.303,-129.978,-78.150,167.685,39.136,157.304
C05174=1034.303,-129.728,-78.163,167.687,39.138,157.305
C05175=1034.304,-129.479,-78.177,167.689,39.140,157.305
C05176=1034.306,-129.228,-78.189,167.691,39.142,157.306
C05177=1034.308,-128.978,-78.200,167.693,39.143,157.306
C05178=1034.311,-128.728,-78.211,167.695,39.144,157.306
C05179=1034.314,-128.478,-78.222,167.698,39.144,157.306
C05180=1034.318,-128.229,-78.232,167.700,39.144,157.306
C05181=1034.323,-127.980,-78.241,167.703,39.143,157.306
C05182=1034.329,-127.730,-78.250,167.706,39.142,157.306
C05183=1034.335,-127.481,-78.259,167.709,39.140,157.306
C05184=1034.342,-127.231,-78.267,167.712,39.139,157.306
C05185=1034.347,-126.981,-78.276,167.714,39.137,157.305
C05186=1034.352,-126.732,-78.285,167.716,39.136,157.305
C05187=1034.359,-126.482,-78.293,167.719,39.135,157.305
C05188=1034.364,-126.232,-78.302,167.722,39.133,157.305
C05189=1034.371,-125.982,-78.310,167.725,39.132,157.305
C05190=1034.376,-125.733,-78.319,167.728,39.131,157.305
C05191=1034.382,-125.482,-78.328,167.731,39.129,157.305
C05192=1034.389,-125.232,-78.336,167.733,39.128,157.304
C05193=1034.394,-124.983,-78.346,167.736,39.127,157.304
C05194=1034.400,-124.733,-78.355,167.739,39.125,157.304
C05195=1034.406,-124.483,-78.362,167.742,39.124,157.304
C05196=1034.412,-124.234,-78.372,167.745,39.123,157.304
C05197=1034.418,-123.984,-78.380,167.748,39.121,157.304
C05198=1034.424,-123.734,-78.390,167.749,39.120,157.304
C05199=1034.430,-123.485,-78.398,167.752,39.119,157.303
C05200=1034.436,-123.234,-78.407,167.755,39.118,157.303
C05201=1034.441,-122.985,-78.416,167.758,39.116,157.303
C05202=1034.447,-122.735,-78.425,167.761,39.115,157.303
C05203=1034.454,-122.485,-78.434,167.764,39.114,157.303
C05204=1034.459,-122.236,-78.442,167.766,39.113,157.303
C05205=1034.466,-121.986,-78.452,167.769,39.111,157.303
C05206=1034.471,-121.736,-78.460,167.772,39.110,157.302
C05207=1034.477,-121.486,-78.469,167.775,39.109,157.302
C05208=1034.484,-121.236,-78.478,167.777,39.107,157.302
C05209=1034.489,-120.986,-78.487,167.780,39.106,157.302
C05210=1034.495,-120.737,-78.496,167.782,39.105,157.302
C05211=1034.500,-120.487,-78.505,167.785,39.103,157.302
C05212=1034.507,-120.237,-78.514,167.788,39.103,157.302
C05213=1034.513,-119.988,-78.523,167.791,39.101,157.302
C05214=1034.519,-119.738,-78.532,167.794,39.100,157.301
C05215=1034.525,-119.488,-78.541,167.797,39.099,157.301
C05216=1034.530,-119.238,-78.550,167.800,39.098,157.301
C05217=1034.537,-118.989,-78.559,167.802,39.096,157.301
C05218=1034.543,-118.738,-78.568,167.804,39.095,157.301
C05219=1034.548,-118.489,-78.577,167.807,39.094,157.301
C05220=1034.555,-118.240,-78.586,167.810,39.092,157.301
C05221=1034.560,-117.989,-78.595,167.813,39.091,157.301
C05222=1034.566,-117.740,-78.604,167.816,39.090,157.300
C05223=1034.572,-117.490,-78.613,167.818,39.089,157.300
C05224=1034.579,-117.240,-78.622,167.821,39.087,157.300
C05225=1034.585,-116.990,-78.632,167.824,39.087,157.300
C05226=1034.591,-116.704,-78.642,167.827,39.085,157.300
C05227=1034.597,-116.417,-78.652,167.830,39.084,157.300
C05228=1034.605,-116.131,-78.663,167.834,39.083,157.300
C05229=1034.612,-115.844,-78.674,167.836,39.081,157.300
C05230=1034.618,-115.595,-78.683,167.839,39.080,157.299
C05231=1034.623,-115.345,-78.692,167.842,39.079,157.299
C05232=1034.629,-115.095,-78.701,167.845,39.077,157.299
C05233=1034.636,-114.846,-78.710,167.847,39.076,157.299
C05234=1034.642,-114.596,-78.720,167.850,39.075,157.299
C05235=1034.648,-114.346,-78.728,167.853,39.074,157.299
C05236=1034.654,-114.096,-78.738,167.855,39.073,157.299
C05237=1034.660,-113.846,-78.747,167.858,39.071,157.299
C05238=1034.666,-113.597,-78.757,167.861,39.071,157.298
C05239=1034.671,-113.347,-78.765,167.864,39.069,157.298
C05240=1034.678,-113.097,-78.775,167.866,39.068,157.298
C05241=1034.684,-112.847,-78.785,167.869,39.067,157.298
C05242=1034.690,-112.598,-78.794,167.872,39.066,157.298
C05243=1034.695,-112.348,-78.803,167.875,39.065,157.298
C05244=1034.701,-112.098,-78.812,167.877,39.063,157.298
C05245=1034.708,-111.848,-78.822,167.880,39.063,157.298
C05246=1034.714,-111.598,-78.831,167.883,39.062,157.298
C05247=1034.720,-111.349,-78.841,167.885,39.060,157.297
C05248=1034.725,-111.100,-78.850,167.888,39.059,157.297
C05249=1034.732,-110.850,-78.860,167.891,39.059,157.297
C05250=1034.737,-110.600,-78.870,167.894,39.057,157.297
C05251=1034.743,-110.350,-78.879,167.896,39.056,157.297
C05252=1034.749,-110.099,-78.888,167.899,39.055,157.297
C05253=1034.755,-109.850,-78.897,167.902,39.054,157.297
C05254=1034.761,-109.601,-78.907,167.904,39.053,157.297
C05255=1034.767,-109.351,-78.917,167.907,39.051,157.297
C05256=1034.773,-109.101,-78.926,167.910,39.051,157.296
C05257=1034.779,-108.851,-78.936,167.913,39.050,157.296
C05258=1034.785,-108.601,-78.945,167.915,39.048,157.296
C05259=1034.792,-108.352,-78.955,167.918,39.047,157.296
C05260=1034.797,-108.102,-78.964,167.921,39.046,157.296
C05261=1034.803,-107.853,-78.974,167.923,39.045,157.296
C05262=1034.810,-107.603,-78.983,167.926,39.044,157.296
C05263=1034.816,-107.353,-78.993,167.929,39.043,157.296
C05264=1034.822,-107.103,-79.002,167.932,39.042,157.296
C05265=1034.827,-106.853,-79.012,167.935,39.041,157.296
C05266=1034.834,-106.603,-79.022,167.938,39.040,157.295
C05267=1034.840,-106.354,-79.032,167.939,39.039,157.295
C05268=1034.845,-106.104,-79.041,167.942,39.038,157.295
C05269=1034.851,-105.855,-79.050,167.945,39.037,157.295
C05270=1034.858,-105.605,-79.060,167.948,39.036,157.295
C05271=1034.863,-105.355,-79.070,167.951,39.035,157.295
C05272=1034.870,-105.106,-79.080,167.954,39.034,157.295
C05273=1034.876,-104.856,-79.090,167.956,39.033,157.295
C05274=1034.882,-104.606,-79.100,167.959,39.032,157.295
C05275=1034.887,-104.356,-79.110,167.961,39.031,157.295
C05276=1034.893,-104.106,-79.119,167.964,39.030,157.295
C05277=1034.900,-103.856,-79.129,167.967,39.029,157.294
C05278=1034.906,-103.606,-79.138,167.969,39.028,157.294
C05279=1034.912,-103.357,-79.149,167.972,39.027,157.294
C05280=1034.918,-103.107,-79.159,167.975,39.026,157.294
C05281=1034.923,-102.858,-79.168,167.978,39.025,157.294
C05282=1034.929,-102.608,-79.178,167.981,39.024,157.294
C05283=1034.936,-102.358,-79.187,167.982,39.023,157.294
C05284=1034.941,-102.109,-79.198,167.985,39.022,157.294
C05285=1034.948,-101.859,-79.208,167.988,39.021,157.294
C05286=1034.954,-101.609,-79.217,167.991,39.020,157.294
C05287=1034.959,-101.359,-79.227,167.994,39.019,157.294
C05288=1034.965,-101.109,-79.237,167.997,39.018,157.293
C05289=1034.972,-100.860,-79.247,167.999,39.017,157.293
C05290=1034.979,-100.573,-79.258,168.003,39.016,157.293
C05291=1034.986,-100.285,-79.270,168.006,39.015,157.293
C05292=1034.993,-99.998,-79.282,168.008,39.014,157.293
C05293=1035.000,-99.711,-79.292,168.011,39.013,157.293
C05294=1035.005,-99.462,-79.303,168.014,39.012,157.293
C05295=1035.012,-99.212,-79.313,168.017,39.011,157.293
C05296=1035.018,-98.962,-79.322,168.020,39.010,157.293
C05297=1035.025,-98.712,-79.333,168.022,39.009,157.293
C05298=1035.030,-98.462,-79.343,168.025,39.008,157.292
C05299=1035.036,-98.213,-79.353,168.028,39.007,157.292
C05300=1035.043,-97.963,-79.363,168.031,39.006,157.292
C05301=1035.048,-97.713,-79.373,168.034,39.006,157.292
C05302=1035.055,-97.463,-79.383,168.035,39.005,157.292
C05303=1035.060,-97.214,-79.394,168.038,39.004,157.292
C05304=1035.066,-96.964,-79.403,168.041,39.003,157.292
C05305=1035.072,-96.715,-79.414,168.044,39.002,157.292
C05306=1035.078,-96.465,-79.424,168.046,39.001,157.292
C05307=1035.084,-96.215,-79.434,168.049,39.000,157.292
C05308=1035.090,-95.966,-79.444,168.052,39.000,157.292
C05309=1035.096,-95.715,-79.454,168.055,38.999,157.292
C05310=1035.102,-95.466,-79.465,168.058,38.998,157.292
C05311=1035.108,-95.216,-79.475,168.060,38.997,157.292
C05312=1035.115,-94.966,-79.485,168.063,38.996,157.291
C05313=1035.120,-94.716,-79.496,168.065,38.995,157.291
C05314=1035.126,-94.467,-79.506,168.068,38.995,157.291
C05315=1035.132,-94.218,-79.517,168.070,38.994,157.291
C05316=1035.138,-93.967,-79.527,168.073,38.993,157.291
C05317=1035.144,-93.718,-79.537,168.076,38.992,157.291
C05318=1035.150,-93.468,-79.547,168.079,38.991,157.291
C05319=1035.156,-93.219,-79.558,168.081,38.990,157.291
C05320=1035.162,-92.969,-79.568,168.084,38.990,157.291
C05321=1035.169,-92.719,-79.578,168.087,38.989,157.291
C05322=1035.174,-92.469,-79.589,168.089,38.989,157.291
C05323=1035.180,-92.219,-79.599,168.092,38.988,157.291
C05324=1035.186,-91.970,-79.610,168.095,38.987,157.291
C05325=1035.192,-91.720,-79.620,168.097,38.986,157.291
C05326=1035.198,-91.471,-79.630,168.099,38.985,157.291
C05327=1035.205,-91.221,-79.641,168.102,38.984,157.291
C05328=1035.211,-90.971,-79.651,168.105,38.983,157.290
C05329=1035.216,-90.721,-79.662,168.108,38.983,157.290
C05330=1035.222,-90.472,-79.673,168.110,38.982,157.290
C05331=1035.228,-90.222,-79.682,168.113,38.981,157.290
C05332=1035.235,-89.972,-79.694,168.116,38.980,157.290
C05333=1035.241,-89.723,-79.704,168.119,38.979,157.290
C05334=1035.247,-89.473,-79.714,168.121,38.979,157.290
C05335=1035.252,-89.223,-79.725,168.124,38.978,157.290
C05336=1035.259,-88.974,-79.735,168.127,38.977,157.290
C05337=1035.265,-88.724,-79.746,168.129,38.977,157.290
C05338=1035.271,-88.474,-79.756,168.131,38.976,157.290
C05339=1035.277,-88.225,-79.767,168.134,38.975,157.290
C05340=1035.283,-87.975,-79.778,168.137,38.974,157.290
C05341=1035.290,-87.725,-79.788,168.140,38.973,157.290
C05342=1035.295,-87.475,-79.799,168.142,38.972,157.290
C05343=1035.302,-87.226,-79.809,168.145,38.972,157.290
C05344=1035.308,-86.976,-79.820,168.148,38.971,157.290
///RCONF 1,0,0,0,0,0,0,0,0,0,0,0,0,0,0,0,0,0,0,0,0,0,0,0
C05345=1035.314,-86.726,-79.831,168.150,38.971,157.290
C05346=1035.320,-86.476,-79.840,168.153,38.970,157.289
C05347=1035.326,-86.227,-79.851,168.156,38.969,157.289
C05348=1035.333,-85.977,-79.862,168.159,38.968,157.289
C05349=1035.339,-85.728,-79.873,168.160,38.967,157.289
C05350=1035.344,-85.478,-79.884,168.163,38.966,157.289
C05351=1035.351,-85.228,-79.894,168.166,38.966,157.289
C05352=1035.357,-84.978,-79.905,168.169,38.965,157.289
C05353=1035.363,-84.729,-79.915,168.171,38.965,157.289
C05354=1035.370,-84.443,-79.928,168.174,38.964,157.289
C05355=1035.377,-84.159,-79.940,168.178,38.963,157.289
C05356=1035.384,-83.874,-79.953,168.181,38.962,157.289
C05357=1035.391,-83.589,-79.965,168.184,38.961,157.289
C05358=1035.398,-83.340,-79.975,168.186,38.960,157.289
C05359=1035.404,-83.090,-79.986,168.189,38.959,157.289
C05360=1035.410,-82.840,-79.997,168.192,38.959,157.289
C05361=1035.416,-82.590,-80.007,168.195,38.958,157.289
C05362=1035.422,-82.340,-80.018,168.196,38.957,157.288
C05363=1035.429,-82.091,-80.028,168.199,38.956,157.288
C05364=1035.435,-81.841,-80.039,168.202,38.956,157.288
C05365=1035.441,-81.591,-80.050,168.205,38.955,157.288
C05366=1035.448,-81.342,-80.061,168.207,38.954,157.288
C05367=1035.454,-81.092,-80.072,168.210,38.953,157.288
C05368=1035.459,-80.843,-80.083,168.213,38.953,157.288
C05369=1035.466,-80.593,-80.093,168.215,38.952,157.288
C05370=1035.472,-80.343,-80.104,168.218,38.951,157.288
C05371=1035.478,-80.093,-80.115,168.221,38.951,157.288
C05372=1035.485,-79.844,-80.126,168.224,38.950,157.288
C05373=1035.491,-79.594,-80.137,168.226,38.949,157.288
C05374=1035.497,-79.344,-80.148,168.229,38.948,157.288
C05375=1035.503,-79.095,-80.159,168.232,38.948,157.288
C05376=1035.509,-78.845,-80.171,168.233,38.947,157.288
C05377=1035.515,-78.596,-80.182,168.236,38.946,157.288
C05378=1035.521,-78.345,-80.193,168.239,38.946,157.288
C05379=1035.527,-78.096,-80.204,168.241,38.945,157.288
C05380=1035.533,-77.846,-80.215,168.244,38.945,157.288
C05381=1035.539,-77.596,-80.226,168.247,38.944,157.288
C05382=1035.546,-77.348,-80.237,168.249,38.944,157.288
C05383=1035.552,-77.098,-80.248,168.252,38.943,157.287
C05384=1035.558,-76.848,-80.259,168.254,38.943,157.288
C05385=1035.564,-76.598,-80.270,168.257,38.942,157.287
C05386=1035.570,-76.348,-80.281,168.260,38.941,157.287
C05387=1035.577,-76.098,-80.292,168.262,38.941,157.287
C05388=1035.583,-75.849,-80.304,168.265,38.940,157.287
C05389=1035.589,-75.599,-80.315,168.268,38.939,157.287
C05390=1035.595,-75.350,-80.326,168.270,38.939,157.287
C05391=1035.601,-75.099,-80.337,168.273,38.938,157.287
C05392=1035.607,-74.851,-80.349,168.276,38.937,157.287
C05393=1035.613,-74.600,-80.360,168.278,38.937,157.287
C05394=1035.619,-74.351,-80.371,168.281,38.936,157.287
C05395=1035.625,-74.101,-80.382,168.283,38.935,157.287
C05396=1035.632,-73.852,-80.394,168.285,38.935,157.287
C05397=1035.638,-73.602,-80.405,168.288,38.935,157.287
C05398=1035.644,-73.352,-80.416,168.291,38.934,157.287
C05399=1035.650,-73.103,-80.428,168.293,38.934,157.287
C05400=1035.656,-72.853,-80.439,168.296,38.933,157.287
C05401=1035.662,-72.603,-80.451,168.298,38.933,157.287
C05402=1035.668,-72.354,-80.462,168.301,38.932,157.287
C05403=1035.674,-72.103,-80.473,168.304,38.932,157.287
C05404=1035.680,-71.855,-80.485,168.306,38.931,157.287
C05405=1035.686,-71.604,-80.496,168.309,38.931,157.287
C05406=1035.692,-71.355,-80.508,168.311,38.930,157.287
C05407=1035.698,-71.105,-80.520,168.314,38.930,157.287
C05408=1035.704,-70.856,-80.531,168.317,38.930,157.287
C05409=1035.710,-70.606,-80.543,168.319,38.929,157.287
C05410=1035.716,-70.357,-80.553,168.322,38.929,157.287
C05411=1035.722,-70.107,-80.566,168.324,38.928,157.287
C05412=1035.728,-69.856,-80.577,168.327,38.928,157.287
C05413=1035.734,-69.608,-80.589,168.330,38.927,157.287
